// TwinCAT 3 PLC project Plc
// Title: CHALET_XPlanar
// Company: Beckhoff CH
// ProjectVersion: 5.8.1
// ProgramVersion: 3.1.4023.0
// libraries:
//   CHALET_BaseComponents, * (Beckhoff CH)
//   CHALET_Nc, * (Beckhoff CH)
//   Tc2_EtherCAT, * (Beckhoff Automation GmbH)
//   Tc2_Math, * (Beckhoff Automation GmbH)
//   Tc2_Standard, * (Beckhoff Automation GmbH)
//   Tc2_System, * (Beckhoff Automation GmbH)
//   Tc2_Utilities, * (Beckhoff Automation GmbH)
//   Tc3_EventLogger, * (Beckhoff Automation GmbH)
//   Tc3_Mc3Definitions, * (Beckhoff Automation GmbH)
//   Tc3_Mc3PlanarMotion, * (Beckhoff Automation GmbH)
//   Tc3_Module, * (Beckhoff Automation GmbH)
//   Tc3_Physics, * (Beckhoff Automation GmbH)
//   Tc3_XPlanarUtility, * (Beckhoff Automation GmbH)
// project tree:
//   COMPONENTs/Environment/ I_XP_Enviroment_PLC.TcIO, FB_XP_Environment.TcPOU, I_XP_Environment.TcIO
//   COMPONENTs/Feedback/ FB_XP_Feedback.TcPOU, I_XP_Feedback.TcIO, ST_PlanarObjectInfoEx.TcDUT
//   COMPONENTs/Mover/ FB_XP_Mover.TcPOU, I_XP_Mover.TcIO, I_XP_Mover_PLC.TcIO
//   COMPONENTs/Mover/ProductData/ FB_XP_ProductData.TcPOU, I_XP_ProductData.TcIO
//   COMPONENTs/Optional/Casting/ ToXpMover.TcPOU, ToXpStation.TcPOU (not stored), ToXpTrack.TcPOU
//   COMPONENTs/Optional/Trigger/ FB_XP_Trigger.TcPOU, I_XP_Trigger.TcIO
//   COMPONENTs/Optional/Zone/ FB_XP_SoretedListOfMover.TcPOU, I_XP_Zone.TcIO
//   COMPONENTs/Path/ FB_XP_Path.TcPOU, I_XP_Path.TcIO
//   COMPONENTs/Stationen/A-Star-Node/ FB_AStarNode.TcPOU, I_PathAStarNode.TcIO
//   COMPONENTs/Stationen/ FB_XP_Station.TcPOU, I_XP_Station.TcIO, I_XP_Station_PLC.TcIO
//   COMPONENTs/Group/ FB_XP_Group.TcPOU, I_XP_Group.TcIO
//   COMPONENTs/System/ FB_XP_System.TcPOU, I_XP_System_PLC.TcIO, I_XP_System_Registration.TcIO
//   COMPONENTs/Track/ FB_XP_Track.TcPOU, I_XP_Track.TcIO, I_XP_Track_PLC.TcIO
//   FUNCTIONs/ F_DistXYVectors.TcPOU, F_Vector_Multiplication.TcPOU, F_Vector_Subtraction.TcPOU, F_GetDistToPosModulo.TcPOU, F_InLimitTest.TcPOU, F_RotatePositionXY.TcPOU, F_Vector_Addition.TcPOU
//   / XPlanarParameterlist.TcGVL

// ---- COMPONENTs/Feedback/ST_PlanarObjectInfoEx.TcDUT
TYPE ST_PlanarObjectInfoEx EXTENDS Tc3_Mc3PlanarMotion.PlanarObjectInfo :
STRUCT
	ipObject : I_CH_Object;
END_STRUCT
END_TYPE

// ---- XPlanarParameterlist.TcGVL
{attribute 'qualified_only'}
VAR_GLOBAL CONSTANT 
	(*After the system init, this is the first station that is approached.
	 Can be used, for example, to send all movers to the “Unload” station first 
	 The default value is “not defined” so the movers remain in the closest station and wait for a valid destination*)
	S_MOVER_TARGED_INIT : STRING := 'not defined';	
	
	(*Only if enabled, mover take over "VelocytiAtExit" of passed station*)	
	B_STATIONS_OVERRIDE_MOVER_DYN_CONSTRAINT : BOOL := FALSE;
	
	(* Automatic generation of missing auxiliary stations on the track. 
	In order to clearly control the route of a mover, for example, when splitting a track into two tracks, an auxiliary station is created on both tracks. 
	The mover must pass this auxiliary station. It moves to it and crosses over as soon as the switch point is passed. 
	This auxiliary station cannot hold a mover (queue size 0) *)
	B_AUTOMATIC_GENARATE_HELPER_STATIONS : BOOL := TRUE;
	
	(*Minimum gap center to center on track [mm] *)
	F_MOVER_MINIMUM_GAP_ON_TRACK : LREAL := 100.0;
	
	(*Default gap center to center on track. Each station can override this gap[mm] *)
	F_GAP_DEFAULT: LREAL := 120.0;
	
	(*Determine the absolute C-rotation of the mover when starting up. Requires an “APM9001-0000-4xxx | XPlanar-ID-Bumper”. *)
	B_GET_MOVER_ORIENTATION : BOOL := FALSE;	
	B_ID_BUMPER_INSTALLED : BOOL := TRUE;
	
	(*Read mover ID when starting up. Requires an “APM9001-0000-4xxx | XPlanar-ID-Bumper”. *)
	B_GET_MOVER_ID : BOOL := FALSE;	
	
	//Quick stop on disable.
	//TRUE = The mover stops immediately AT the current position
	//FALSE = The mover cancels the superimposed ExternalSetpoint movement and returns to the track with maximum dynamic. -> Like a rubber band
	B_QUICKSTOP_ON_DISABLING : BOOL := TRUE;
	
	//When the system is enabled, the system checks which movers are actually present. 
	//Any movers that are not present are moved forward to the “NotPresent” list
	B_AUTOMATICALLY_REMOVE_NOT_PRESENT_MOVER_AT_ENABLING : BOOL := TRUE;	
	
	(*Add envirement to groupe during enabling *)
	B_ADD_ENVIROMENT_TO_GROUP : BOOL := TRUE;	
					
	(*Add tracks to groupe during enabling *)
	B_ADD_TRACKS_TO_GROUP : BOOL := FALSE;	
					
	(*Add movers to groupe during enabling *)
	B_ADD_MOVERS_TO_GROUP : BOOL := FALSE;	
					
	//Velocity during enabling move on track. 0=Default
	F_ENABLING_ON_TRACK_VELOCITY	: LREAL := 0;
	
	(*Acc-/Deceleration during enabling move on track. 0=Default*)
	F_ENABLING_ON_TRACK_ACC_DEC		: LREAL := 0;
	
	(*This value as a Station.Filter allows all movers of any target*)
	S_ANY_STATION_NAME : STRING := '';
	
	//TRUE = Use inside PLC the track name from the TcCom Track Object. If FALSE overwride TcCom Track object with instance name
	B_TRACK_NAME_TACKOVER_FROM_TRACK_OBJECT : BOOL := TRUE;
	
	//If a single-cell sequence step takes longer than this time when enabling the entire system, an error is generated and the enabling is aborted
	F_TIMEOUT_ERROR_ENABLING : LREAL := 30.0; //[s]
	
	(*The movers are only sent to the next free station on the way to the destination. 
	The distance in mm can be specified here to indicate how much further away the new move command can already be sent.  *)
	F_DIST_SET_NEW_MOVE_CMD_BEFORE_REACHING_PARENT_STATION : LREAL := 200.0;
	
	(*max tracks after a track switch *)
	N_MAX_STATIONS_AHEAD_OR_BEHIND : UINT := 20;	
	
	(*A mover must leave the station immediately when the ‘SendMoversToStation’ method is called. The station is then available again.
	Otherwise, if no destination station is available, the mover waits in the station.*)
	B_MOVER_MUST_LEAVE_STATION_AT_SET_NEW_TARGED : BOOL := TRUE;
	
	(*0: Indicates no or invalid information, e.g. no connection or component not yet ready. 
	1: The Planar Mover interprets the given dynamic limits in a one-dimensional fashion, with respect to the track's arclength. This way, the maximum velocity is aimed at even in curves. 
	2: The maximal velocity in curves is reduced to not exceed the maximum x,y radial acceleration there. Produces the same behavior as the None mode when on a straight track. 	*)
	N_SELECT_MODE_HOW_DYNAMIC_IS_PLANED_ON_TRACK : UINT := 2;
	
	(*Indicates the way in which gap control is done on track.
	1:The Planar Mover keeps a distance to its neighbours on track that is at least the sum of gap and stop distance.
	2:The Planar Mover keeps a distance to its neighbours on track that is at least the gap.*)
	N_GAP_MODE_ON_TRACK : UINT := 2;
	
	(* How many elements (point, line or arc) does the most complex track have? *)
	N_MAX_GEOMETRIC_ELEMENTS_PER_TRACK : UINT := 20;
END_VAR

// ---- COMPONENTs/Environment/I_XP_Enviroment_PLC.TcIO
INTERFACE I_XP_Enviroment_PLC EXTENDS I_CH_Object

{attribute 'monitoring':='call'}
(* If Enable, the movers are checked for collisions with each other.
Warning and error can have their own size offsets.
The error leads to a stop with higher dynamics.
In simulation, an error does not lead to a stop *)
PROPERTY CollisionCheck : BOOL
GET
END_GET
SET
END_SET
END_PROPERTY

{attribute 'monitoring':='call'}
//Offset on the mover dimension from the MC3 mover object [mm] ;
// >0 menas the warning is earlier
PROPERTY MoverCollisionOffsetError : LREAL
GET
END_GET
SET
END_SET
END_PROPERTY

{attribute 'monitoring':='call'}
//Offset on the mover dimension from the MC3 mover object [mm] ;
// >0 menas the warning is earlier
PROPERTY MoverCollisionOffsetWarning : LREAL
GET
END_GET
SET
END_SET
END_PROPERTY

{attribute 'monitoring':='call'}
//Enumeration MoverDetectionStatus
PROPERTY MoverDetectionStatus : MoverDetectionStatus
GET
END_GET
END_PROPERTY

{attribute 'monitoring':='call'}
//Object ID of the IoXPlanar processing unit
PROPERTY ProcessingUnitOID : OTCID
GET
END_GET
END_PROPERTY

{attribute 'monitoring':='call'}
//Interface to CHALET system to which this object belongs
PROPERTY System : I_XP_System_PLC
GET
END_GET
END_PROPERTY

END_INTERFACE

// ---- COMPONENTs/Feedback/I_XP_Feedback.TcIO
INTERFACE I_XP_Feedback EXTENDS CHALET_BaseComponents.I_CH_Feedback

{attribute 'monitoring':='call'}
(* Indicates which object one would collide with. *)
PROPERTY ObjectInfo : REFERENCE TO PlanarObjectInfo
GET
END_GET
SET
END_SET
END_PROPERTY

{attribute 'monitoring':='call'}
(* Indicates which object one would collide with. *)
PROPERTY ObjectInfoEx : REFERENCE TO ST_PlanarObjectInfoEx
GET
END_GET
SET
END_SET
END_PROPERTY

END_INTERFACE

// ---- COMPONENTs/Mover/I_XP_Mover.TcIO
INTERFACE I_XP_Mover  EXTENDS I_CH_Object

{attribute 'monitoring':='call'}
(* Provides the current planar mover setpoint XYZABC [mm/s²] *)
PROPERTY AccelerationSet : REFERENCE TO MoverVector
GET
END_GET
END_PROPERTY

METHOD AddToGroup : HRESULT
VAR_INPUT
	iGroup : I_XP_Group;
END_VAR
END_METHOD

{attribute 'monitoring':='call'}
(* C coordinate modulus set in MC3-Planar Mover[°] *)
PROPERTY CAxisModulo : LREAL
GET
END_GET
END_PROPERTY

{attribute 'monitoring':='call'}
PROPERTY CurrentTrack : I_XP_Track
GET
END_GET
END_PROPERTY

METHOD Disable : HRESULT
VAR_INPUT
END_VAR
END_METHOD

//This method is called when the system is disabled. Links are deleted as they may no longer be valid
METHOD Disassemble : HRESULT
VAR_INPUT
END_VAR
END_METHOD

{attribute 'monitoring':='call'}
PROPERTY DistToParentStation : LREAL //Distance to the responsible parent station [mm]
GET
END_GET
END_PROPERTY

METHOD DistToTrack : LREAL
VAR_INPUT
	iTrack : I_XP_Track;
END_VAR
END_METHOD

PROPERTY DynConstraint : REFERENCE TO DynamicConstraint_Container
GET
END_GET
END_PROPERTY

METHOD Enable : HRESULT
VAR_INPUT
END_VAR
END_METHOD

{attribute 'monitoring':='call'}
//operational and position control active(hovering)
PROPERTY Enabled : BOOL
GET
END_GET
END_PROPERTY

{attribute 'OPC.UA.DA.Property' := '1'}
{attribute 'monitoring':='call'}
PROPERTY Feedback : I_XP_Feedback
GET
END_GET
END_PROPERTY

METHOD Halt : HRESULT
VAR_INPUT
END_VAR
END_METHOD

METHOD JoinTrack : HRESULT
VAR_INPUT
	iTrack : I_XP_Track;
END_VAR
END_METHOD

{attribute 'monitoring':='call'}
PROPERTY LastCmdTargetGap : LREAL
GET
END_GET
END_PROPERTY

{attribute 'monitoring':='call'}
PROPERTY LastCmdTargetPosition : LREAL
GET
END_GET
END_PROPERTY

{attribute 'monitoring':='call'}
PROPERTY LastCmdTargetTrack: I_XP_Track
GET
END_GET
END_PROPERTY

{attribute 'monitoring':='call'}
//This was the last valid (system enabled) parent station of the mover
PROPERTY LastValidParentStation : I_XP_Station;
GET
END_GET
END_PROPERTY

{attribute 'monitoring':='call'}
//This was the last valid (system enabled) actual  position of the mover
PROPERTY LastValidPositionOnTrack : LREAL
GET
END_GET
END_PROPERTY

{attribute 'monitoring':='call'}
//This was the last valid (system enabled) actual  position of the mover
PROPERTY LastValidPositionXYZABC : REFERENCE TO MoverVector
GET
END_GET
END_PROPERTY

{attribute 'monitoring':='call'}
//This was the last valid (system enabled) actual  position of the mover
PROPERTY LastValidTrack : I_XP_Track;
GET
END_GET
END_PROPERTY

//The mover returns to its SetPos. The force of the Z, A and B axis is slowly increased.
METHOD LiftFromUnknownLevel : HRESULT
VAR_INPUT
END_VAR
END_METHOD

(* The mover is lowered. The target height is unknown. The force from the Z, A and B axles is then reduced to a minimum. X, Y and C still remain active.
   This function can be used, for example, to place the mover in a holder.  *)
METHOD LowerToUnknownLevel : HRESULT
VAR_INPUT
END_VAR
END_METHOD

{attribute 'monitoring':='call'}
PROPERTY Mapped : BOOL //Project is mapped to MC (McToPlc and PlcToMc)
GET
END_GET
END_PROPERTY

{attribute 'monitoring':='call'}
PROPERTY Mode : MC_PLANAR_MOVER_COMMAND_MODE
GET
END_GET
END_PROPERTY

METHOD MoveA : HRESULT
VAR_INPUT
	fPosition : LREAL;
END_VAR
END_METHOD

METHOD MoveB : HRESULT
VAR_INPUT
	fPosition : LREAL;
END_VAR
END_METHOD

METHOD MoveC : HRESULT
VAR_INPUT
	fPosition : LREAL;
	
	(* Addition turns to move in modulo movement (positive or negative). *)
	additionalTurns : UDINT := 0;
	
	(* Direction in which the target is approached. *)
	direction : Tc3_Mc3Definitions.MC_DIRECTION := Tc3_Mc3Definitions.MC_DIRECTION.mcDirectionNonModulo;
END_VAR
END_METHOD

METHOD MoveOnTrack : HRESULT
VAR_INPUT
	ipTrack : I_XP_Track;
	fPosition : LREAL;
	fGap : LREAL;
END_VAR
END_METHOD

METHOD MoveOnTrack_ShortestWay : HRESULT
VAR_INPUT
	ipTrack : I_XP_Track;
	fPosition : LREAL;
	fGap : LREAL;
END_VAR
END_METHOD

METHOD MoveOnTrackToStation : HRESULT
VAR_INPUT
	ipStation : I_XP_Station;
	fGap : LREAL;
END_VAR
END_METHOD

{attribute 'monitoring':='call'}
(* Height that is used for internal collision checks.[mm] *)
PROPERTY MoverHeight : LREAL
GET
END_GET
END_PROPERTY

{attribute 'monitoring':='call'}
//Mover could not be detected or was removed from the system
PROPERTY MoverIsNotPresent : BOOL
GET
END_GET
END_PROPERTY

{attribute 'monitoring':='call'}
(* Width that is used for internal collision checks.[mm] *)
PROPERTY MoverWidth : LREAL
GET
END_GET
END_PROPERTY

METHOD MoveXY : HRESULT
VAR_INPUT
	fPosition_X : LREAL;
	fPosition_Y : LREAL;
END_VAR
END_METHOD

METHOD MoveZ : HRESULT
VAR_INPUT
	fPosition : LREAL;
END_VAR
END_METHOD

{attribute 'monitoring':='call'}
//Unique object ID
PROPERTY OID : OTCID
GET
END_GET
END_PROPERTY

{attribute 'monitoring':='call'}
PROPERTY ParentStation : I_XP_Station
GET
END_GET
SET
END_SET
END_PROPERTY

{attribute 'monitoring':='call'}
PROPERTY PlanarMover : REFERENCE TO MC_PlanarMover
GET
END_GET
END_PROPERTY

{attribute 'monitoring':='call'}
(* Contains the information of the Planar Mover passed from MC to PLC. XYZABC [mm] *)
PROPERTY PositionAct : REFERENCE TO MoverVector
GET
END_GET
END_PROPERTY

{attribute 'monitoring':='call'}
PROPERTY PositionOnTrack : LREAL
GET
END_GET
END_PROPERTY

{attribute 'monitoring':='call'}
(* Provides the current planar mover setpoint XYZABC [mm] *)
PROPERTY PositionSet : REFERENCE TO MoverVector
GET
END_GET
END_PROPERTY

METHOD RemoveFromGroup : HRESULT
END_METHOD

METHOD Reset : HRESULT
VAR_INPUT
END_VAR
END_METHOD

{attribute 'monitoring':='call'}
//Complete route from last parent to active parent station
PROPERTY RouteComplete : I_CH_List
GET
END_GET
END_PROPERTY

{attribute 'monitoring':='call'}
//Remaining route to the parent
PROPERTY RouteRemaining: I_CH_List
GET
END_GET
END_PROPERTY

//done segments can be transferred here. these are removed from the remaining route
METHOD RouteSegmentDone : BOOL
VAR_INPUT
	ipPathDone : I_XP_Path;
END_VAR
END_METHOD

METHOD SetDynConstraint_A : BOOL //Dynamic constraints for individual coordinates.
VAR_INPUT
    V : MC_LREAL; //equivalent to data type LREAL + MC_DEFAULT, MC_MAXIMUM
    A : MC_LREAL; //equivalent to data type LREAL + MC_DEFAULT, MC_MAXIMUM
    D : MC_LREAL; //equivalent to data type LREAL + MC_DEFAULT, MC_MAXIMUM
    J : MC_LREAL; //equivalent to data type LREAL + MC_DEFAULT, MC_MAXIMUM
END_VAR
END_METHOD

METHOD SetDynConstraint_B : BOOL //Dynamic constraints for individual coordinates.
VAR_INPUT
    V : MC_LREAL; //equivalent to data type LREAL + MC_DEFAULT, MC_MAXIMUM
    A : MC_LREAL; //equivalent to data type LREAL + MC_DEFAULT, MC_MAXIMUM
    D : MC_LREAL; //equivalent to data type LREAL + MC_DEFAULT, MC_MAXIMUM
    J : MC_LREAL; //equivalent to data type LREAL + MC_DEFAULT, MC_MAXIMUM
END_VAR
END_METHOD

METHOD SetDynConstraint_C : BOOL //Dynamic constraints for individual coordinates.
VAR_INPUT
    V : MC_LREAL; //equivalent to data type LREAL + MC_DEFAULT, MC_MAXIMUM
    A : MC_LREAL; //equivalent to data type LREAL + MC_DEFAULT, MC_MAXIMUM
    D : MC_LREAL; //equivalent to data type LREAL + MC_DEFAULT, MC_MAXIMUM
    J : MC_LREAL; //equivalent to data type LREAL + MC_DEFAULT, MC_MAXIMUM
END_VAR
END_METHOD

METHOD SetDynConstraint_Path : BOOL //One dimensional dynamic constraint along the XY-components of a path, ignoring non-tangential effects.
VAR_INPUT
    V : MC_LREAL; //equivalent to data type LREAL + MC_DEFAULT, MC_MAXIMUM
    A : MC_LREAL; //equivalent to data type LREAL + MC_DEFAULT, MC_MAXIMUM
    D : MC_LREAL; //equivalent to data type LREAL + MC_DEFAULT, MC_MAXIMUM
    J : MC_LREAL; //equivalent to data type LREAL + MC_DEFAULT, MC_MAXIMUM
END_VAR
END_METHOD

METHOD SetDynConstraint_X : BOOL //Dynamic constraints for individual coordinates.
VAR_INPUT
    V : MC_LREAL; //equivalent to data type LREAL + MC_DEFAULT, MC_MAXIMUM
    A : MC_LREAL; //equivalent to data type LREAL + MC_DEFAULT, MC_MAXIMUM
    D : MC_LREAL; //equivalent to data type LREAL + MC_DEFAULT, MC_MAXIMUM
    J : MC_LREAL; //equivalent to data type LREAL + MC_DEFAULT, MC_MAXIMUM
END_VAR
END_METHOD

METHOD SetDynConstraint_Y : BOOL //Dynamic constraints for individual coordinates.
VAR_INPUT
    V : MC_LREAL; //equivalent to data type LREAL + MC_DEFAULT, MC_MAXIMUM
    A : MC_LREAL; //equivalent to data type LREAL + MC_DEFAULT, MC_MAXIMUM
    D : MC_LREAL; //equivalent to data type LREAL + MC_DEFAULT, MC_MAXIMUM
    J : MC_LREAL; //equivalent to data type LREAL + MC_DEFAULT, MC_MAXIMUM
END_VAR
END_METHOD

METHOD SetDynConstraint_Z : BOOL //Dynamic constraints for individual coordinates.
VAR_INPUT
    V : MC_LREAL; //equivalent to data type LREAL + MC_DEFAULT, MC_MAXIMUM
    A : MC_LREAL; //equivalent to data type LREAL + MC_DEFAULT, MC_MAXIMUM
    D : MC_LREAL; //equivalent to data type LREAL + MC_DEFAULT, MC_MAXIMUM
    J : MC_LREAL; //equivalent to data type LREAL + MC_DEFAULT, MC_MAXIMUM
END_VAR
END_METHOD

METHOD SetRouteToParent : HRESULT
VAR_INPUT
	ipRoute : I_CH_LIST;
END_VAR
END_METHOD

{attribute 'monitoring':='call'}
(* Velocity is zero *)
PROPERTY Standstill : BOOL
GET
END_GET
END_PROPERTY

METHOD StopExternalSetpoint : HRESULT
VAR_INPUT
END_VAR
END_METHOD

{attribute 'monitoring':='call'}
PROPERTY TargetStation : String
GET
END_GET
SET
END_SET
END_PROPERTY

{attribute 'monitoring':='call'}
PROPERTY UtilityMcMover : Tc3_XPlanarUtility.I_McPlanarMover
GET
END_GET
END_PROPERTY

PROPERTY UtilityTcIoMover : Tc3_XPlanarUtility.I_TcIoXPlanarMover
GET
END_GET
END_PROPERTY

{attribute 'monitoring':='call'}
(* Provides the current planar mover act XYZABC [mm/s] *)
PROPERTY VelocityAct : REFERENCE TO MoverVector
GET
END_GET
END_PROPERTY

{attribute 'monitoring':='call'}
(* Provides the current planar mover setpoint XYZABC [mm/s] *)
PROPERTY VelocitySet : REFERENCE TO MoverVector
GET
END_GET
END_PROPERTY

END_INTERFACE

// ---- COMPONENTs/Mover/I_XP_Mover_PLC.TcIO
INTERFACE I_XP_Mover_PLC EXTENDS I_CH_Object

{attribute 'monitoring':='call'}
(* Provides the current planar mover setpoint XYZABC [mm/s²] *)
PROPERTY AccelerationSet : REFERENCE TO MoverVector
GET
END_GET
END_PROPERTY

{attribute 'monitoring':='call'}
PROPERTY  AxisExtSetpointA : CHALET_Nc.I_NcAxis_PLC
GET
END_GET
END_PROPERTY

{attribute 'monitoring':='call'}
PROPERTY AxisExtSetpointB : CHALET_Nc.I_NcAxis_PLC
GET
END_GET
END_PROPERTY

{attribute 'monitoring':='call'}
PROPERTY AxisExtSetpointC : CHALET_Nc.I_NcAxis_PLC
GET
END_GET
END_PROPERTY

{attribute 'monitoring':='call'}
PROPERTY  AxisExtSetpointX : CHALET_Nc.I_NcAxis_PLC
GET
END_GET
END_PROPERTY

{attribute 'monitoring':='call'}
PROPERTY AxisExtSetpointY : CHALET_Nc.I_NcAxis_PLC
GET
END_GET
END_PROPERTY

{attribute 'monitoring':='call'}
PROPERTY AxisExtSetpointZ : CHALET_Nc.I_NcAxis_PLC
GET
END_GET
END_PROPERTY

{attribute 'monitoring':='call'}
(* C coordinate modulus set in MC3-Planar Mover[°] *)
PROPERTY CAxisModulo : LREAL
GET
END_GET
END_PROPERTY

{attribute 'monitoring':='call'}
(* Indicates the command mode of an enabled PlanarMover, i.e. how setpoints are currently produced. *)
PROPERTY CommandMode : MC_PLANAR_MOVER_COMMAND_MODE
GET
END_GET
END_PROPERTY

{attribute 'monitoring':='call'}
PROPERTY CurrentTrack : I_XP_Track
GET
END_GET
END_PROPERTY

{attribute 'monitoring':='call'}
PROPERTY DistToParentStation : LREAL //Distance to the responsible parent station [mm]
GET
END_GET
END_PROPERTY

METHOD DistToTrack : LREAL
VAR_INPUT
	iTrack : I_XP_Track;
END_VAR
END_METHOD

PROPERTY DynConstraint : REFERENCE TO DynamicConstraint_Container
GET
END_GET
END_PROPERTY

{attribute 'monitoring':='call'}
//operational and position control active(hovering)
PROPERTY Enabled : BOOL
GET
END_GET
END_PROPERTY

{attribute 'OPC.UA.DA.Property' := '1'}
{attribute 'monitoring':='call'}
PROPERTY Feedback : I_XP_Feedback
GET
END_GET
END_PROPERTY

METHOD Halt : HRESULT
VAR_INPUT
END_VAR
END_METHOD

METHOD JoinTrack : HRESULT
VAR_INPUT
	iTrack : I_XP_Track;
END_VAR
END_METHOD

{attribute 'monitoring':='call'}
(* Retruns lentgh of hypotenuse of the x and y error. (>=0[mm]) *)
PROPERTY LagDistanceXY : LREAL
GET
END_GET
END_PROPERTY

{attribute 'monitoring':='call'}
PROPERTY LastCmdTargetGap : LREAL
GET
END_GET
END_PROPERTY

{attribute 'monitoring':='call'}
PROPERTY LastCmdTargetPosition : LREAL
GET
END_GET
END_PROPERTY

{attribute 'monitoring':='call'}
PROPERTY LastCmdTargetTrack: I_XP_Track
GET
END_GET
END_PROPERTY

{attribute 'monitoring':='call'}
//This was the last valid (system enabled) parent station of the mover
PROPERTY LastValidParentStation : I_XP_Station;
GET
END_GET
END_PROPERTY

{attribute 'monitoring':='call'}
//This was the last valid (system enabled) actual  position of the mover
PROPERTY LastValidPositionOnTrack : LREAL
GET
END_GET
END_PROPERTY

{attribute 'monitoring':='call'}
//This was the last valid (system enabled) actual  position of the mover
PROPERTY LastValidPositionXYZABC : REFERENCE TO MoverVector
GET
END_GET
END_PROPERTY

{attribute 'monitoring':='call'}
//This was the last valid (system enabled) actual  position of the mover
PROPERTY LastValidTrack : I_XP_Track;
GET
END_GET
END_PROPERTY

//The mover returns to its SetPos. The force of the Z, A and B axis is slowly increased.
METHOD LiftFromUnknownLevel : HRESULT
VAR_INPUT
END_VAR
END_METHOD

(* The mover is lowered. The target height is unknown. The force from the Z, A and B axles is then reduced to a minimum. X, Y and C still remain active.
   This function can be used, for example, to place the mover in a holder.  *)
METHOD LowerToUnknownLevel : HRESULT
VAR_INPUT
END_VAR
END_METHOD

{attribute 'monitoring':='call'}
PROPERTY LUID : STRING //Locally unique identifier
GET
END_GET
END_PROPERTY

{attribute 'monitoring':='call'}
PROPERTY Mapped : BOOL //Project is mapped to MC (McToPlc and PlcToMc)
GET
END_GET
END_PROPERTY

METHOD MoveA : HRESULT
VAR_INPUT
	fPosition : LREAL;
END_VAR
END_METHOD

METHOD MoveB : HRESULT
VAR_INPUT
	fPosition : LREAL;
END_VAR
END_METHOD

METHOD MoveC : HRESULT
VAR_INPUT
	fPosition : LREAL;
	
	(* Addition turns to move in modulo movement (positive or negative). *)
	additionalTurns : UDINT := 0;
	
	(* Direction in which the target is approached. *)
	direction : Tc3_Mc3Definitions.MC_DIRECTION := Tc3_Mc3Definitions.MC_DIRECTION.mcDirectionNonModulo;
END_VAR
END_METHOD

METHOD MoveOnTrack : HRESULT
VAR_INPUT
	ipTrack : I_XP_Track;
	fPosition : LREAL;
	fGap : LREAL;
END_VAR
END_METHOD

METHOD MoveOnTrack_ShortestWay : HRESULT
VAR_INPUT
	ipTrack : I_XP_Track;
	fPosition : LREAL;
	fGap : LREAL;
END_VAR
END_METHOD

{attribute 'monitoring':='call'}
(* Height that is used for internal collision checks.[mm] *)
PROPERTY MoverHeight : LREAL
GET
END_GET
END_PROPERTY

{attribute 'monitoring':='call'}
//Mover could not be detected or was removed from the system
PROPERTY MoverIsNotPresent : BOOL
GET
END_GET
END_PROPERTY

{attribute 'monitoring':='call'}
(* Width that is used for internal collision checks.[mm] *)
PROPERTY MoverWidth : LREAL
GET
END_GET
END_PROPERTY

METHOD MoveXY : HRESULT
VAR_INPUT
	fPosition_X : LREAL;
	fPosition_Y : LREAL;
END_VAR
END_METHOD

METHOD MoveZ : HRESULT
VAR_INPUT
	fPosition : LREAL;
END_VAR
END_METHOD

{attribute 'monitoring':='call'}
//Unique object ID
PROPERTY OID : OTCID
GET
END_GET
END_PROPERTY

{attribute 'monitoring':='call'}
PROPERTY ParentStation : I_XP_Station
GET
END_GET
END_PROPERTY

{attribute 'monitoring':='call'}
PROPERTY PlanarMover : REFERENCE TO MC_PlanarMover
GET
END_GET
END_PROPERTY

{attribute 'monitoring':='call'}
(* Contains the information of the Planar Mover passed from MC to PLC. XYZABC [mm] *)
PROPERTY PositionAct : REFERENCE TO MoverVector
GET
END_GET
END_PROPERTY

{attribute 'monitoring':='call'}
PROPERTY PositionOnTrack : LREAL
GET
END_GET
END_PROPERTY

{attribute 'monitoring':='call'}
(* Provides the current planar mover setpoint XYZABC [mm] *)
PROPERTY PositionSet : REFERENCE TO MoverVector
GET
END_GET
END_PROPERTY

{attribute 'monitoring':='call'}
PROPERTY PUBLIC ProductData : I_XP_ProductData
GET
END_GET
SET
END_SET
END_PROPERTY

{attribute 'monitoring':='call'}
//Complete route from last parent to active parent station
PROPERTY RouteComplete : I_CH_List
GET
END_GET
END_PROPERTY

{attribute 'monitoring':='call'}
//Remaining route to the parent
PROPERTY RouteRemaining: I_CH_List
GET
END_GET
END_PROPERTY

//done segments can be transferred here. these are removed from the remaining route
METHOD RouteSegmentDone : BOOL
VAR_INPUT
	ipPathDone : I_XP_Path;
END_VAR
END_METHOD

METHOD SetDynConstraint_A : BOOL //Dynamic constraints for individual coordinates.
VAR_INPUT
    V : MC_LREAL; //equivalent to data type LREAL + MC_DEFAULT, MC_MAXIMUM
    A : MC_LREAL; //equivalent to data type LREAL + MC_DEFAULT, MC_MAXIMUM
    D : MC_LREAL; //equivalent to data type LREAL + MC_DEFAULT, MC_MAXIMUM
    J : MC_LREAL; //equivalent to data type LREAL + MC_DEFAULT, MC_MAXIMUM
END_VAR
END_METHOD

METHOD SetDynConstraint_B : BOOL //Dynamic constraints for individual coordinates.
VAR_INPUT
    V : MC_LREAL; //equivalent to data type LREAL + MC_DEFAULT, MC_MAXIMUM
    A : MC_LREAL; //equivalent to data type LREAL + MC_DEFAULT, MC_MAXIMUM
    D : MC_LREAL; //equivalent to data type LREAL + MC_DEFAULT, MC_MAXIMUM
    J : MC_LREAL; //equivalent to data type LREAL + MC_DEFAULT, MC_MAXIMUM
END_VAR
END_METHOD

METHOD SetDynConstraint_C : BOOL //Dynamic constraints for individual coordinates.
VAR_INPUT
    V : MC_LREAL; //equivalent to data type LREAL + MC_DEFAULT, MC_MAXIMUM
    A : MC_LREAL; //equivalent to data type LREAL + MC_DEFAULT, MC_MAXIMUM
    D : MC_LREAL; //equivalent to data type LREAL + MC_DEFAULT, MC_MAXIMUM
    J : MC_LREAL; //equivalent to data type LREAL + MC_DEFAULT, MC_MAXIMUM
END_VAR
END_METHOD

METHOD SetDynConstraint_Path : BOOL //One dimensional dynamic constraint along the XY-components of a path, ignoring non-tangential effects.
VAR_INPUT
    V : MC_LREAL; //equivalent to data type LREAL + MC_DEFAULT, MC_MAXIMUM
    A : MC_LREAL; //equivalent to data type LREAL + MC_DEFAULT, MC_MAXIMUM
    D : MC_LREAL; //equivalent to data type LREAL + MC_DEFAULT, MC_MAXIMUM
    J : MC_LREAL; //equivalent to data type LREAL + MC_DEFAULT, MC_MAXIMUM
END_VAR
END_METHOD

METHOD SetDynConstraint_X : BOOL //Dynamic constraints for individual coordinates.
VAR_INPUT
    V : MC_LREAL; //equivalent to data type LREAL + MC_DEFAULT, MC_MAXIMUM
    A : MC_LREAL; //equivalent to data type LREAL + MC_DEFAULT, MC_MAXIMUM
    D : MC_LREAL; //equivalent to data type LREAL + MC_DEFAULT, MC_MAXIMUM
    J : MC_LREAL; //equivalent to data type LREAL + MC_DEFAULT, MC_MAXIMUM
END_VAR
END_METHOD

METHOD SetDynConstraint_Y : BOOL //Dynamic constraints for individual coordinates.
VAR_INPUT
    V : MC_LREAL; //equivalent to data type LREAL + MC_DEFAULT, MC_MAXIMUM
    A : MC_LREAL; //equivalent to data type LREAL + MC_DEFAULT, MC_MAXIMUM
    D : MC_LREAL; //equivalent to data type LREAL + MC_DEFAULT, MC_MAXIMUM
    J : MC_LREAL; //equivalent to data type LREAL + MC_DEFAULT, MC_MAXIMUM
END_VAR
END_METHOD

METHOD SetDynConstraint_Z : BOOL //Dynamic constraints for individual coordinates.
VAR_INPUT
    V : MC_LREAL; //equivalent to data type LREAL + MC_DEFAULT, MC_MAXIMUM
    A : MC_LREAL; //equivalent to data type LREAL + MC_DEFAULT, MC_MAXIMUM
    D : MC_LREAL; //equivalent to data type LREAL + MC_DEFAULT, MC_MAXIMUM
    J : MC_LREAL; //equivalent to data type LREAL + MC_DEFAULT, MC_MAXIMUM
END_VAR
END_METHOD

METHOD SetRouteToParent : HRESULT
VAR_INPUT
	ipRoute : I_CH_LIST;
END_VAR
END_METHOD

{attribute 'monitoring':='call'}
(* Velocity is zero *)
PROPERTY Standstill : BOOL
GET
END_GET
END_PROPERTY

METHOD StartExternalSetpoint : HRESULT
END_METHOD

METHOD StopExternalSetpoint : HRESULT
VAR_INPUT
END_VAR
END_METHOD

{attribute 'monitoring':='call'}
//Interface to CHALET system to which this object belongs
PROPERTY System : I_XP_System_PLC
GET
END_GET
END_PROPERTY

{attribute 'monitoring':='call'}
PROPERTY TargetStation : STRING
GET
END_GET
SET
END_SET
END_PROPERTY

{attribute 'monitoring':='call'}
PROPERTY UtilityMcMover : Tc3_XPlanarUtility.I_McPlanarMover
GET
END_GET
END_PROPERTY

{attribute 'monitoring':='call'}
PROPERTY UtilityTcIoMover : Tc3_XPlanarUtility.I_TcIoXPlanarMover
GET
END_GET
END_PROPERTY

{attribute 'monitoring':='call'}
(* Provides the current planar mover act XYZABC [mm/s] *)
PROPERTY VelocityAct : REFERENCE TO MoverVector
GET
END_GET
END_PROPERTY

{attribute 'monitoring':='call'}
(* Provides the current planar mover setpoint XYZABC [mm/s] *)
PROPERTY VelocitySet : REFERENCE TO MoverVector
GET
END_GET
END_PROPERTY

END_INTERFACE

// ---- COMPONENTs/Mover/ProductData/I_XP_ProductData.TcIO
INTERFACE I_XP_ProductData EXTENDS __SYSTEM.IQueryInterface

{attribute 'monitoring':='call'}
PROPERTY LinkedMover : I_XP_Mover_PLC
GET
END_GET
END_PROPERTY

METHOD LinkToMover : BOOL //it is not necessary to call this method. This is already done internally
VAR_INPUT
	ipMoverPlc : I_XP_Mover_PLC;
END_VAR
END_METHOD

END_INTERFACE

// ---- COMPONENTs/Optional/Trigger/I_XP_Trigger.TcIO
INTERFACE I_XP_Trigger  EXTENDS __SYSTEM.IQueryInterface

{attribute 'monitoring':='call'}
PROPERTY AccocietedTrack : I_XP_Track
GET
END_GET
SET
END_SET
END_PROPERTY

{attribute 'monitoring':='call'}
PROPERTY HR : HRESULT
GET
END_GET
END_PROPERTY

PROPERTY ListOfMoversToCheck : I_CH_List
SET
END_SET
END_PROPERTY

{attribute 'monitoring':='call'}
PROPERTY MoverAtTrigger : I_XP_Mover
GET
END_GET
END_PROPERTY

{attribute 'monitoring':='call'}
PROPERTY MoverDetected : BOOL
GET
END_GET
END_PROPERTY

{attribute 'monitoring':='call'}
PROPERTY PositionOnTrack : LREAL
GET
END_GET
SET
END_SET
END_PROPERTY

{attribute 'monitoring':='call'}
PROPERTY TimeStamp : T_DCTIME64;
GET
END_GET
END_PROPERTY

{attribute 'monitoring':='call'}
PROPERTY TriggerDirection : Tc3_Mc3Definitions.MC_Direction
GET
END_GET
SET
END_SET
END_PROPERTY

END_INTERFACE

// ---- COMPONENTs/Optional/Zone/I_XP_Zone.TcIO
INTERFACE I_XP_Zone

{attribute 'monitoring':='call'}
PROPERTY CtsMoversInZone : UINT
GET
END_GET
END_PROPERTY

{attribute 'monitoring':='call'}
PROPERTY MoversInZone : REFERENCE TO ARRAY [0..(CHALET_BaseComponents.BaseParameterlist.MAX_OBJECTS-1)] OF I_XP_Mover_PLC // Return a sorted list of movers in this zone. Index 0 is the mover in Front.
GET
END_GET
END_PROPERTY

END_INTERFACE

// ---- COMPONENTs/Path/I_XP_Path.TcIO
INTERFACE I_XP_Path  EXTENDS I_CH_Object

METHOD DistanceToDestiantion : LREAL
VAR_INPUT
	ipTrack : I_XP_Track;
	fPosOnTrack : LREAL;
END_VAR
END_METHOD

{attribute 'monitoring':='call'}
PROPERTY Length : LREAL
GET
END_GET
SET
END_SET
END_PROPERTY

{attribute 'monitoring':='call'}
PROPERTY StationDestination : I_XP_Station
GET
END_GET
SET
END_SET
END_PROPERTY

{attribute 'monitoring':='call'}
PROPERTY StationStart  : I_XP_Station
GET
END_GET
SET
END_SET
END_PROPERTY

{attribute 'monitoring':='call'}
PROPERTY TracksUsed : REFERENCE TO FB_CH_List
GET
END_GET
END_PROPERTY

END_INTERFACE

// ---- COMPONENTs/Stationen/A-Star-Node/I_PathAStarNode.TcIO
INTERFACE I_PathAStarNode EXTENDS I_CH_Object

{attribute 'monitoring':='call'}
PROPERTY PathLength : LREAL
GET
END_GET
END_PROPERTY

{attribute 'monitoring':='call'}
PROPERTY RouteUsedToNode : REFERENCE TO FB_CH_List
GET
END_GET
END_PROPERTY

{attribute 'monitoring':='call'}
PROPERTY Station : I_XP_Station
GET
END_GET
SET
END_SET
END_PROPERTY

END_INTERFACE

// ---- COMPONENTs/Stationen/I_XP_Station.TcIO
INTERFACE I_XP_Station EXTENDS I_CH_Object

{attribute 'monitoring':='call'}
//Track on which the station is located
PROPERTY AccocietedTrack : I_XP_Track
GET
END_GET
END_PROPERTY

METHOD AddMoverToQueue : HRESULT
VAR_INPUT
	ipMover : I_XP_Mover;
END_VAR
END_METHOD

{attribute 'monitoring':='call'}
//List of movers managed by this station
PROPERTY AssignedMovers : I_CH_List
GET
END_GET
END_PROPERTY

//Call this Methode whith seq 0->100, and wait each step until S_OK is returned
METHOD Configure : HRESULT
VAR_INPUT
	nSeq : UINT; //0->100
END_VAR
END_METHOD

{attribute 'monitoring':='call'}
PROPERTY CtsEmptySpaceInQueue : UDINT
GET
END_GET
END_PROPERTY

{attribute 'monitoring':='call'}
PROPERTY CtsMoversInQueue : UDINT
GET
END_GET
END_PROPERTY

{attribute 'monitoring':='call'}
(*[mm]
As soon as the mover is closer than this distance, the mover can be sent on to the next one if necessary.
This is the distance from the station to the end of the track or the shortest path to this station. Depending on which is closer. This is to ensure that the mover can no longer be overhauled.
This proberty can make the internal calculated distance smaller but not larger
Recalculated each disable/enable of the system*)
PROPERTY DecisionDistance : LREAL
GET
END_GET
SET
END_SET
END_PROPERTY

METHOD DeleteMoversQueue : HRESULT
VAR_INPUT
END_VAR
END_METHOD

//This method is called when the system is disabled. Links are deleted as they may no longer be valid
METHOD Disassemble : HRESULT
VAR_INPUT
END_VAR
END_METHOD

{attribute 'monitoring':='call'}
PROPERTY Filter : STRING
GET
END_GET
SET
END_SET
END_PROPERTY

{attribute 'monitoring':='call'}
PROPERTY MoverAccAtExit : MC_LREAL //[mm/s² on Track] Every mover that leaves or passes the station gets this new acceleration as a target.
GET
END_GET
END_PROPERTY

{attribute 'monitoring':='call'}
PROPERTY MoverDecAtExit : MC_LREAL //[mm/s² on Track] Every mover that leaves or passes the station gets this new deceleration as a target.
GET
END_GET
END_PROPERTY

{attribute 'monitoring':='call'}
//[mm] Every mover that leaves or passes the station gets this new gap as a target.
PROPERTY MoverGapAtExit : LREAL
GET
END_GET
SET
END_SET
END_PROPERTY

{attribute 'monitoring':='call'}
PROPERTY MoverQueueSize : UINT
GET
END_GET
END_PROPERTY

{attribute 'monitoring':='call'}
PROPERTY MoversInPlace : BOOL
GET
END_GET
END_PROPERTY

{attribute 'monitoring':='call'}
PROPERTY MoverVelocityAtExit : MC_LREAL //[mm/s on Track] Every mover that leaves or passes the station gets this new velocity as a target.
GET
END_GET
END_PROPERTY

{attribute 'monitoring':='call'}
//List of paths that lead to stations before this station
PROPERTY PathsAhead : I_CH_List
GET
END_GET
END_PROPERTY

{attribute 'monitoring':='call'}
//List of paths that lead to stations behind this station
PROPERTY PathsBehinde : I_CH_List
GET
END_GET
END_PROPERTY

{attribute 'monitoring':='call'}
//[mm] from the beginning of the assigned track
PROPERTY PositionOnTrack : LREAL
GET
END_GET
END_PROPERTY

{attribute 'monitoring':='call'}
//Position on the assigned track
PROPERTY PositionOnTrackXY : REFERENCE TO PositionXY
GET
END_GET
END_PROPERTY

{attribute 'monitoring':='call'}
//Position on the assigned track
PROPERTY PositionOnTrackXYZABC : REFERENCE TO MoverVector
GET
END_GET
END_PROPERTY

{attribute 'monitoring':='call'}
//Planned position, not necessarily on the track
PROPERTY PositionXY : REFERENCE TO  PositionXY
GET
END_GET
END_PROPERTY

//The movers currently in this station must leave the station. 
//The movers actively search for a destination, but only leave if a new destination is available.
METHOD PushMoversOutOfStation : HRESULT
VAR_INPUT
END_VAR
END_METHOD

{attribute 'monitoring':='call'}
//prevent further movers from entering the station, 
//e.g. to prevent a collision. All movers that are already moving to reach this station will be stopped with a stop 
//and restarted with Ready True.
PROPERTY ReadyToRecvMovers : BOOL
GET
END_GET
END_PROPERTY

METHOD SendMoversToStation : I_CH_Feedback //All movers in the station are sent to this destination
VAR_INPUT
	sTargetStation: STRING;//unique station name or group of stations
END_VAR
END_METHOD

{attribute 'monitoring':='call'}
//List of stations before this station
PROPERTY StationsAhead : I_CH_List
GET
END_GET
END_PROPERTY

{attribute 'monitoring':='call'}
//List of stations behinde this station
PROPERTY StationsBehinde : I_CH_List
GET
END_GET
END_PROPERTY

{attribute 'monitoring':='call'}
PROPERTY TargetGroupe : STRING
GET
END_GET
END_PROPERTY

METHOD Update : HRESULT
VAR_INPUT
END_VAR
END_METHOD

END_INTERFACE

// ---- COMPONENTs/Stationen/I_XP_Station_PLC.TcIO
INTERFACE I_XP_Station_PLC EXTENDS I_CH_Object

{attribute 'monitoring':='call'}
//Track on which the station is located
PROPERTY AccocietedTrack : I_XP_Track
GET
END_GET
END_PROPERTY

{attribute 'monitoring':='call'}
PROPERTY CtsEmptySpaceInQueue : UDINT
GET
END_GET
END_PROPERTY

{attribute 'monitoring':='call'}
PROPERTY CtsMoversInQueue : UDINT
GET
END_GET
END_PROPERTY

{attribute 'monitoring':='call'}
(*[mm]
As soon as the mover is closer than this distance, the mover can be sent on to the next one if necessary.
This is the distance from the station to the end of the track or the shortest path to this station. Depending on which is closer. This is to ensure that the mover can no longer be overhauled.
This proberty can make the internal calculated distance smaller but not larger
Recalculated each disable/enable of the system*)
PROPERTY DecisionDistance : LREAL
GET
END_GET
SET
END_SET
END_PROPERTY

{attribute 'monitoring':='call'}
PROPERTY Feedback : I_CH_Feedback
GET
END_GET
END_PROPERTY

{attribute 'monitoring':='call'}
//Filter content, movers with one of these targets may not approach or drive over the station
PROPERTY Filter : STRING
GET
END_GET
SET
END_SET
END_PROPERTY

{attribute 'monitoring':='call'}
PROPERTY LUID : STRING //Locally unique identifier
GET
END_GET
END_PROPERTY

{attribute 'monitoring':='call'}
PROPERTY MoverAccAtExit : MC_LREAL //[mm/s² on Track] Every mover that leaves or passes the station gets this new acceleration as a target.
GET
END_GET
SET
END_SET
END_PROPERTY

{attribute 'monitoring':='call'}
PROPERTY MoverDecAtExit : MC_LREAL //[mm/s² on Track] Every mover that leaves or passes the station gets this new deceleration as a target.
GET
END_GET
SET
END_SET
END_PROPERTY

{attribute 'monitoring':='call'}
PROPERTY MoverGapAtExit : LREAL //[mm] Every mover that leaves or passes the station gets this new gap as a target.
GET
END_GET
SET
END_SET
END_PROPERTY

{attribute 'monitoring':='call'}
PROPERTY MoverQueueSize : UINT
GET
END_GET
SET
END_SET
END_PROPERTY

{attribute 'monitoring':='call'}
PROPERTY MoversInPlace : BOOL
GET
END_GET
END_PROPERTY

{attribute 'monitoring':='call'}
PROPERTY MoversInQueue : REFERENCE TO ARRAY [0..(CHALET_BaseComponents.BaseParameterlist.MAX_OBJECTS-1)] OF I_XP_Mover_PLC // Return a sorted list of movers in this zone. Index 0 is the mover in Front
GET
END_GET
END_PROPERTY

{attribute 'monitoring':='call'}
PROPERTY MoverVelocityAtExit : MC_LREAL //[mm/s on Track] Every mover that leaves or passes the station gets this new velocity as a target.
GET
END_GET
SET
END_SET
END_PROPERTY

{attribute 'monitoring':='call'}
//[mm] from the beginning of the assigned track
PROPERTY PositionOnTrack : LREAL
GET
END_GET
END_PROPERTY

{attribute 'monitoring':='call'}
//Position on the assigned track
PROPERTY PositionOnTrackXY : REFERENCE TO PositionXY
GET
END_GET
END_PROPERTY

{attribute 'monitoring':='call'}
//Planned position, not necessarily on the track
PROPERTY PositionXY : REFERENCE TO  PositionXY
GET
END_GET
END_PROPERTY

{attribute 'monitoring':='call'}
PROPERTY ProcessSimulationActive : BOOL
GET
END_GET
END_PROPERTY

//The movers currently in this station must leave the station. 
//The movers actively search for a destination, but only leave if a new destination is available.
METHOD PushMoversOutOfStation : HRESULT
VAR_INPUT
END_VAR
END_METHOD

{attribute 'monitoring':='call'}
//prevent further movers from entering the station, 
//e.g. to prevent a collision. All movers that are already moving to reach this station will be stopped with a stop 
//and restarted with Ready True.
PROPERTY ReadyToRecvMovers : BOOL
GET
END_GET
SET
END_SET
END_PROPERTY

METHOD SendMoversToStation : I_CH_Feedback //All movers in the station are sent to this destination
VAR_INPUT
	sTargetStation: STRING;//unique station name or group of stations
END_VAR
END_METHOD

//If a valid time (>0seconds) is set and the configured destination station exists, then the movers will be sent away automatically after this time from now on.
METHOD SimulationStart : HRESULT
VAR_INPUT
	fProcessDuration 		: LREAL; //[s]
	sTargetStation	: STRING; //Group of the target station to automatic send after the duration
END_VAR
END_METHOD

//If a valid time (>0seconds) is set and the configured destination station exists, then the movers will be sent away automatically after this time from now on.
METHOD SimulationStartEx : HRESULT
VAR_INPUT
	fProcessDuration 		: LREAL; //[s]
	ipStation				: I_XP_Station_PLC; //unique station to automatic send after the duration
END_VAR
END_METHOD

METHOD SimulationStop : HRESULT
END_METHOD

{attribute 'monitoring':='call'}
//List of stations before this station
PROPERTY StationsAhead : I_CH_List
GET
END_GET
END_PROPERTY

{attribute 'monitoring':='call'}
//List of stations behinde this station
PROPERTY StationsBehinde : I_CH_List
GET
END_GET
END_PROPERTY

{attribute 'monitoring':='call'}
//Suppress to change the dynamic(Gap+velocity) of passing movers. This is usefull in startup
PROPERTY SuppressDynamicsChange : BOOL
GET
END_GET
SET
END_SET
END_PROPERTY

{attribute 'monitoring':='call'}
//Interface to CHALET system to which this object belongs
PROPERTY System : I_XP_System_PLC
GET
END_GET
END_PROPERTY

{attribute 'monitoring':='call'}
PROPERTY TargetGroupe : STRING
GET
END_GET
END_PROPERTY

{attribute 'monitoring':='call'}
//A time that is waited as soon as the mover is in the station (including the monitoring window) before “MoversInPlace” is set. e.g. used to stabilize the workpiece
PROPERTY TargetPosMonitoringTime : TIME
GET
END_GET
SET
END_SET
END_PROPERTY

{attribute 'monitoring':='call'}
//How many mm before the mover reaches the position is “MoversInPlace” set for the process. 
//This distance can also be set very large (e.g. 100mm) for moving past without stopping.
PROPERTY TargetPosWindow : LREAL
GET
END_GET
SET
END_SET
END_PROPERTY

END_INTERFACE

// ---- COMPONENTs/Environment/I_XP_Environment.TcIO
INTERFACE I_XP_Environment EXTENDS I_CH_Object

METHOD AddToGroup : HRESULT
VAR_INPUT
	iGroup : I_XP_Group;
END_VAR
END_METHOD

(* Clears the Planar Environment (stators and boundary). *)
METHOD Clear : HRESULT
END_METHOD

METHOD Configure : HRESULT
VAR_INPUT
END_VAR
END_METHOD

{attribute 'monitoring':='call'}
PROPERTY Feedback : I_XP_Feedback
GET
END_GET
END_PROPERTY

METHOD Initialize : HRESULT
END_METHOD

{attribute 'monitoring':='call'}
PROPERTY Mapped : BOOL //Project is mapped to MC (McToPlc and PlcToMc)
GET
END_GET
END_PROPERTY

{attribute 'monitoring':='call'}
//Unique object ID
PROPERTY OID : OTCID
GET
END_GET
END_PROPERTY

{attribute 'monitoring':='call'}
PROPERTY PlanarEnvironment : REFERENCE TO MC_PlanarEnvironment
GET
END_GET
END_PROPERTY

{attribute 'monitoring':='call'}
//Enumeration MoverDetectionStatus
PROPERTY ProcessingUnitMoverDetectionStatus : MoverDetectionStatus
GET
END_GET
END_PROPERTY

{attribute 'monitoring':='call'}
//Object ID of the IoXPlanar processing unit
PROPERTY ProcessingUnitOID : OTCID
GET
END_GET
END_PROPERTY

METHOD RemoveFromGroup : HRESULT
END_METHOD

METHOD PUBLIC Update : HRESULT
VAR_INPUT
END_VAR
END_METHOD

{attribute 'monitoring':='call'}
PROPERTY UtilityEnvirement : Tc3_XPlanarUtility.I_Environment
GET
END_GET
END_PROPERTY

END_INTERFACE

// ---- COMPONENTs/Group/I_XP_Group.TcIO
INTERFACE I_XP_Group  EXTENDS I_CH_Object

METHOD AddEnvironment : HRESULT
VAR_INPUT
	refEnvironment : REFERENCE TO MC_PlanarEnvironment;
	refFeedback : REFERENCE TO MC_PlanarFeedback;
END_VAR
END_METHOD

METHOD AddMover : HRESULT
VAR_INPUT
	refMover : REFERENCE TO MC_PlanarMover;
	refFeedback : REFERENCE TO MC_PlanarFeedback;
END_VAR
END_METHOD

METHOD AddTrack : HRESULT
VAR_INPUT
	refTrack : REFERENCE TO MC_PlanarTrack;
	refFeedback : REFERENCE TO MC_PlanarFeedback;
END_VAR
END_METHOD

METHOD Disable : HRESULT
VAR_INPUT
END_VAR
END_METHOD

METHOD Enable : HRESULT
VAR_INPUT
END_VAR
END_METHOD

{attribute 'OPC.UA.DA.Property' := '1'}
{attribute 'monitoring':='call'}
PROPERTY Feedback : I_XP_Feedback
GET
END_GET
END_PROPERTY

METHOD Initialize : HRESULT
VAR_INPUT
END_VAR
END_METHOD

{attribute 'monitoring':='call'}
PROPERTY Mapped : BOOL //Project is mapped to MC (McToPlc and PlcToMc)
GET
END_GET
END_PROPERTY

{attribute 'monitoring':='call'}
//Unique object ID
PROPERTY OID : OTCID
GET
END_GET
END_PROPERTY

{attribute 'monitoring':='call'}
PROPERTY PlanarGroup : REFERENCE TO MC_PlanarGroup
GET
END_GET
END_PROPERTY

METHOD Reset : HRESULT
VAR_INPUT
END_VAR
END_METHOD

METHOD PUBLIC Update : HRESULT
VAR_INPUT
END_VAR
END_METHOD

END_INTERFACE

// ---- COMPONENTs/System/I_XP_System_PLC.TcIO
INTERFACE I_XP_System_PLC EXTENDS I_CH_Object

METHOD CheckTargetExists : BOOL //Return TRUE if target is existing
VAR_INPUT
	sStation	: STRING; //Group of the target station or LUID
END_VAR
END_METHOD

METHOD Disable : I_CH_Feedback
VAR_INPUT
END_VAR
END_METHOD

{attribute 'monitoring':='call'}
PROPERTY Disabled : BOOL
GET
END_GET
END_PROPERTY

METHOD Enable : I_CH_Feedback
VAR_INPUT
END_VAR
END_METHOD

{attribute 'monitoring':='call'}
PROPERTY Enabled : BOOL
GET
END_GET
END_PROPERTY

{attribute 'monitoring':='call'}
PROPERTY Enviroment : I_XP_Environment
GET
END_GET
END_PROPERTY

METHOD FastStop : I_CH_Feedback
END_METHOD

{attribute 'monitoring':='call'}
PROPERTY Feedback : CHALET_BaseComponents.I_CH_Feedback
GET
END_GET
END_PROPERTY

//Returns the station that is closest to the point according to Phytagoras
METHOD GetStationClosestTo : I_XP_Station
VAR_INPUT
	pos : MoverVector;
END_VAR
END_METHOD

METHOD Initialize : HRESULT
VAR_INPUT
END_VAR
END_METHOD

{attribute 'monitoring':='call'}
PROPERTY Initialized : BOOL
GET
END_GET
END_PROPERTY

{attribute 'monitoring':='call'}
//List of movers that are not present in the current system
PROPERTY MoversNotPresent : CHALET_BaseComponents.I_CH_LIST
GET
END_GET
END_PROPERTY

{attribute 'monitoring':='call'}
//List of movers that are present in the current system
PROPERTY MoversPresent : CHALET_BaseComponents.I_CH_LIST
GET
END_GET
END_PROPERTY

{attribute 'monitoring':='call'}
PROPERTY Paths : CHALET_BaseComponents.I_CH_LIST
GET
END_GET
END_PROPERTY

METHOD Station : I_XP_Station_PLC
VAR_INPUT
	sLUID : STRING;
END_VAR
END_METHOD

{attribute 'monitoring':='call'}
//List of all station objects that exist in this project
PROPERTY StationsAll : CHALET_BaseComponents.I_CH_LIST
GET
END_GET
END_PROPERTY

{attribute 'monitoring':='call'}
//List of all station objects that are considered for path planning in the currently running system
PROPERTY StationsUsed : CHALET_BaseComponents.I_CH_LIST
GET
END_GET
END_PROPERTY

//Suppress to change the dynamic(Gap) of passing movers in all stations. This is usefull in startup
PROPERTY SuppressAllDynamicsChanges : BOOL
SET
END_SET
END_PROPERTY

{attribute 'monitoring':='call'}
PROPERTY Tracks : CHALET_BaseComponents.I_CH_LIST
GET
END_GET
END_PROPERTY

{attribute 'monitoring':='call'}
PROPERTY Triggers : CHALET_BaseComponents.I_CH_LIST
GET
END_GET
END_PROPERTY

METHOD Update : HRESULT
VAR_INPUT
END_VAR
END_METHOD

{attribute 'monitoring':='call'}
PROPERTY Zones : CHALET_BaseComponents.I_CH_LIST
GET
END_GET
END_PROPERTY

END_INTERFACE

// ---- COMPONENTs/System/I_XP_System_Registration.TcIO
INTERFACE I_XP_System_Registration EXTENDS __SYSTEM.IQueryInterface

{attribute 'monitoring':='call'}
PROPERTY Disabled : BOOL
GET
END_GET
END_PROPERTY

{attribute 'monitoring':='call'}
PROPERTY Enabled : BOOL
GET
END_GET
END_PROPERTY

{attribute 'monitoring':='call'}
PROPERTY Enviroment : I_XP_Environment
GET
END_GET
END_PROPERTY

METHOD LinkEnvironment : HRESULT
VAR_INPUT
	ipEnvironment : I_CH_Object;
END_VAR
END_METHOD

METHOD LinkGroup : HRESULT
VAR_INPUT
	ipGroup : I_CH_Object;
END_VAR
END_METHOD

{attribute 'monitoring':='call'}
//List of movers that are not present in the current system
PROPERTY MoversNotPresent : CHALET_BaseComponents.I_CH_LIST
GET
END_GET
END_PROPERTY

{attribute 'monitoring':='call'}
//List of movers that are present in the current system
PROPERTY MoversPresent : CHALET_BaseComponents.I_CH_LIST
GET
END_GET
END_PROPERTY

{attribute 'monitoring':='call'}
PROPERTY Paths : CHALET_BaseComponents.I_CH_LIST
GET
END_GET
END_PROPERTY

METHOD RegisterMover : HRESULT
VAR_INPUT
	ipMover : I_CH_Object;
END_VAR
END_METHOD

METHOD RegisterStation : HRESULT
VAR_INPUT
	ipStation : I_CH_Object;
END_VAR
END_METHOD

METHOD RegisterTrack : HRESULT
VAR_INPUT
	ipTrack : I_CH_Object;
END_VAR
END_METHOD

METHOD RegisterTrigger : HRESULT
VAR_INPUT
	ipTrigger	: CHALET_BaseComponents.I_CH_Object;
END_VAR
END_METHOD

METHOD RegisterZone : HRESULT
VAR_INPUT
	ipZone	: CHALET_BaseComponents.I_CH_Object;
END_VAR
END_METHOD

{attribute 'monitoring':='call'}
//List of all station objects that exist in this project
PROPERTY StationsAll : CHALET_BaseComponents.I_CH_LIST
GET
END_GET
END_PROPERTY

{attribute 'monitoring':='call'}
//List of all station objects that are considered for path planning in the currently running system
PROPERTY StationsUsed : CHALET_BaseComponents.I_CH_LIST
GET
END_GET
END_PROPERTY

{attribute 'monitoring':='call'}
PROPERTY Tracks : CHALET_BaseComponents.I_CH_LIST
GET
END_GET
END_PROPERTY

{attribute 'monitoring':='call'}
PROPERTY Triggers : CHALET_BaseComponents.I_CH_LIST
GET
END_GET
END_PROPERTY

{attribute 'monitoring':='call'}
PROPERTY Zones : CHALET_BaseComponents.I_CH_LIST
GET
END_GET
END_PROPERTY

END_INTERFACE

// ---- COMPONENTs/Track/I_XP_Track.TcIO
INTERFACE I_XP_Track  EXTENDS I_CH_Object

METHOD AddMover : HRESULT
VAR_INPUT
	ipMover : I_XP_Mover;
END_VAR
END_METHOD

METHOD AddToGroup : HRESULT
VAR_INPUT
	iGroup : I_XP_Group;
END_VAR
END_METHOD

{attribute 'monitoring':='call'}
PROPERTY ClosedLoop : BOOL
GET
END_GET
END_PROPERTY

METHOD Configure : HRESULT
VAR_INPUT
END_VAR
END_METHOD

METHOD Configuring : HRESULT
VAR_INPUT
END_VAR
END_METHOD

{attribute 'monitoring':='call'}
PROPERTY CtsMoversOnTrack : UINT
GET
END_GET
END_PROPERTY

METHOD Disable : HRESULT
VAR_INPUT
END_VAR
END_METHOD

METHOD Enable : HRESULT
VAR_INPUT
END_VAR
END_METHOD

{attribute 'monitoring':='call'}
//Position of the end point of this tracks
PROPERTY EndPosition : REFERENCE TO MoverVector
GET
END_GET
END_PROPERTY

{attribute 'monitoring':='call'}
PROPERTY Feedback : I_XP_Feedback
GET
END_GET
END_PROPERTY

(* Calculates which gap the mover should have on a position
	The gap results from the last station crossed.
	If several stations are possible ( switch), the largest gap is displayed here *)
METHOD GapAtPosition : LREAL
VAR_INPUT
	fPosOnTrack : LREAL;//[mm]	
END_VAR
END_METHOD

//Each track has an auxiliary station at the end of itself. This is used automatically or not, depending on whether the track also contains stations created by the user.
//These are used by the movers as auxiliary links to navigate through a complex network.
{attribute 'monitoring':='call'}
PROPERTY HelperStationAtEndOfTrack : I_XP_Station
GET
END_GET
END_PROPERTY

{attribute 'monitoring':='call'}
//[mm]
PROPERTY Length : LREAL
GET
END_GET
END_PROPERTY

{attribute 'monitoring':='call'}
PROPERTY PlanarTrack : REFERENCE TO MC_PlanarTrack
GET
END_GET
END_PROPERTY

METHOD RemoveFromGroup : HRESULT
END_METHOD

METHOD Reset : HRESULT
VAR_INPUT
END_VAR
END_METHOD

{attribute 'monitoring':='call'}
//Position of the start point of this tracks
PROPERTY StartPosition : REFERENCE TO MoverVector
GET
END_GET
END_PROPERTY

(* Returns the first station on current track who has exact thsi position or is ahead
	If no station on this track, result is maybe on another track*)
METHOD StationAhedPosition : I_XP_Station
VAR_INPUT
	fPosOnTrack : LREAL;//[mm]	
END_VAR
END_METHOD

(* Returns the first station on current track who has exact this position or is behind
	If no station on this track, result is maybe on another track*)
METHOD StationBehindPosition : I_XP_Station
VAR_INPUT
	fPosOnTrack : LREAL;//[mm]	
END_VAR
END_METHOD

(* Returns the closest station on current, ahead or behind track*)
METHOD StationClosestTo : I_XP_Station
VAR_INPUT
	fPosOnTrack : LREAL;//[mm]	
END_VAR
END_METHOD

{attribute 'monitoring':='call'}
//List of interfaces to stations on this track
PROPERTY StationsOnTrack : I_CH_List
GET
END_GET
END_PROPERTY

{attribute 'monitoring':='call'}
//List of interfaces from other tracks
PROPERTY TracksAhead : I_CH_List
GET
END_GET
END_PROPERTY

{attribute 'monitoring':='call'}
//List of interfaces from other tracks
PROPERTY TracksBehinde : I_CH_List
GET
END_GET
END_PROPERTY

{attribute 'monitoring':='call'}
PROPERTY TracksEndAtThis : REFERENCE TO  ARRAY[0..(XPlanarParameterlist.N_MAX_STATIONS_AHEAD_OR_BEHIND-1)] OF I_XP_Track
GET
END_GET
END_PROPERTY

{attribute 'monitoring':='call'}
PROPERTY TracksStartFromThis : REFERENCE TO ARRAY[0..(XPlanarParameterlist.N_MAX_STATIONS_AHEAD_OR_BEHIND-1)] OF I_XP_Track
GET
END_GET
END_PROPERTY

{attribute 'monitoring':='call'}
//Interface to this track in XPlanar Utility Lib
PROPERTY UtilityTrack : Tc3_XPlanarUtility.I_McPlanarTrack
GET
END_GET
END_PROPERTY

END_INTERFACE

// ---- COMPONENTs/Track/I_XP_Track_PLC.TcIO
INTERFACE I_XP_Track_PLC EXTENDS I_CH_Object

{attribute 'monitoring':='call'}
PROPERTY CtsMoversOnTrack : UINT
GET
END_GET
END_PROPERTY

{attribute 'monitoring':='call'}
//Position of the end point of this tracks
PROPERTY EndPosition : REFERENCE TO MoverVector
GET
END_GET
END_PROPERTY

{attribute 'monitoring':='call'}
PROPERTY Feedback : I_XP_Feedback
GET
END_GET
END_PROPERTY

{attribute 'monitoring':='call'}
//[mm]
PROPERTY Length : LREAL
GET
END_GET
END_PROPERTY

{attribute 'monitoring':='call'}
PROPERTY Mapped : BOOL //Project is mapped to MC (McToPlc and PlcToMc)
GET
END_GET
END_PROPERTY

{attribute 'monitoring':='call'}
// Number of elements describing the geometric curve of the track.
PROPERTY NbOfGeometricElements : UINT
GET
END_GET
END_PROPERTY

{attribute 'monitoring':='call'}
//Unique object ID
PROPERTY OID : OTCID
GET
END_GET
END_PROPERTY

{attribute 'monitoring':='call'}
PROPERTY PlanarTrack : REFERENCE TO MC_PlanarTrack
GET
END_GET
END_PROPERTY

//The geometric points of a track are copied. Including the position and type. This only works if the system is disabled.
METHOD ReplicateGeometricElements : HRESULT
VAR_INPUT
	ipTrackCopyFrom : I_XP_Track;
END_VAR
END_METHOD

//move all points of the track geometry. Only works if the system is disabled.
METHOD ShiftTrack : HRESULT
VAR_INPUT
	xOffset, yOffset : LREAL;
END_VAR
END_METHOD

{attribute 'monitoring':='call'}
//Position of the start point of this tracks
PROPERTY StartPosition : REFERENCE TO MoverVector
GET
END_GET
END_PROPERTY

(* Returns the first station on current track who has exact thsi position or is ahead
	If no station on this track, result is maybe on another track*)
METHOD StationAhedPosition : I_XP_Station
VAR_INPUT
	fPosOnTrack : LREAL;//[mm]	
END_VAR
END_METHOD

(* Returns the first station on current track who has exact thsi position or is behind
	If no station on this track, result is maybe on another track*)
METHOD StationBehindPosition : I_XP_Station
VAR_INPUT
	fPosOnTrack : LREAL;//[mm]	
END_VAR
END_METHOD

(* Returns the closest station on current, ahead or behind track*)
METHOD StationClosestTo : I_XP_Station
VAR_INPUT
	fPosOnTrack : LREAL;//[mm]	
END_VAR
END_METHOD

{attribute 'monitoring':='call'}
//List of interfaces to stations on this track
PROPERTY StationsOnTrack : I_CH_List
GET
END_GET
END_PROPERTY

{attribute 'monitoring':='call'}
//Interface to CHALET system to which this object belongs
PROPERTY System : I_XP_System_PLC
GET
END_GET
END_PROPERTY

{attribute 'monitoring':='call'}
//List of interfaces from other tracks
PROPERTY TracksAhead : I_CH_List
GET
END_GET
END_PROPERTY

{attribute 'monitoring':='call'}
//List of interfaces from other tracks
PROPERTY TracksBehinde : I_CH_List
GET
END_GET
END_PROPERTY

{attribute 'monitoring':='call'}
PROPERTY TracksEndAtThis : REFERENCE TO  ARRAY[0..(XPlanarParameterlist.N_MAX_STATIONS_AHEAD_OR_BEHIND-1)] OF I_XP_Track
GET
END_GET
END_PROPERTY

{attribute 'monitoring':='call'}
PROPERTY TracksStartFromThis : REFERENCE TO ARRAY[0..(XPlanarParameterlist.N_MAX_STATIONS_AHEAD_OR_BEHIND-1)] OF I_XP_Track
GET
END_GET
END_PROPERTY

{attribute 'monitoring':='call'}
//Interface to this track in XPlanar Utility Lib
PROPERTY UtilityTrack : Tc3_XPlanarUtility.I_McPlanarTrack
GET
END_GET
END_PROPERTY

END_INTERFACE

// ---- COMPONENTs/Feedback/FB_XP_Feedback.TcPOU
{attribute 'no_explicit_call' := 'Do not call the body - Stick to OOP'}
FUNCTION_BLOCK FB_XP_Feedback EXTENDS CHALET_Nc.FB_NcFeedback IMPLEMENTS I_XP_Feedback
VAR_INPUT
END_VAR
VAR_OUTPUT
END_VAR
VAR
	(* Indicates which object one would collide with. *)
	{attribute 'hide'}
	_objectInfo : ST_PlanarObjectInfoEx;
END_VAR

METHOD ClearObjectInfo : BOOL
VAR_INPUT
END_VAR
THIS^._ObjectInfo.Id := 0;
THIS^._ObjectInfo.ipObject := 0;
THIS^._ObjectInfo.ObjectType := EPlanarObjectType.None;
END_METHOD

{attribute 'monitoring':='call'}
(* Indicates which object one would collide with. *)
PROPERTY ObjectInfo : REFERENCE TO PlanarObjectInfo
GET
objectInfo REF= THIS^._objectInfo;
END_GET
SET
THIS^._objectInfo.Id			:= ObjectInfo.Id;
THIS^._objectInfo.ObjectType 	:= ObjectInfo.ObjectType;
THIS^._objectInfo.ipObject 		:= 0;
END_SET
END_PROPERTY

{attribute 'monitoring':='call'}
(* Indicates which object one would collide with. *)
PROPERTY ObjectInfoEx : REFERENCE TO ST_PlanarObjectInfoEx
GET
objectInfoEx REF= THIS^._objectInfo;
END_GET
SET
THIS^._objectInfo := ObjectInfoEx;
END_SET
END_PROPERTY

END_FUNCTION_BLOCK

// ---- COMPONENTs/Mover/FB_XP_Mover.TcPOU
// The warning " Interface of overridden methode xxx of base I_xxx doesn't match declaration" can be disabled here. 
{warning disable C0094 }
{attribute 'no_explicit_call' := 'Do not call the body - Stick to OOP'}
(* XPlanar mover - n per associated XPlanar. Can be instantiated as an array and/or individually
	The Planar mover is a software object that represents an XPlanar mover. It summarizes the state of the real mover (position, velocity, etc.) 
	for the user. In addition, the user has the possibility to influence or control the state of the real mover via the Planar mover. *)	
FUNCTION_BLOCK FB_XP_Mover EXTENDS FB_CH_Object IMPLEMENTS I_XP_Mover, I_XP_Mover_PLC
VAR
	fbRouteRemaining : FB_CH_List;//Remaining route to the parent station
	fbRouteComplete : FB_CH_List;//Complete route from last parent to active parent station
END_VAR

VAR
	//Link to MC-Mover
	fbMover : MC_PlanarMover; 
	
	{attribute 'hide'}  
	bInitDone :BOOL := FALSE;
	{attribute 'hide'}               	
	fbFeedback 			: FB_XP_Feedback(ipSourceInfo := fbSourceInfo);	
	{attribute 'hide'}                   	
	eActiveCommand 		: CHALET_Nc.E_NcAxisCommands := CHALET_Nc.E_NcAxisCommands.None;
	{attribute 'hide'}
	ipXpSystem : I_XP_System_Registration;
	{attribute 'hide'} 
	sTargetStation : STRING := XPlanarParameterlist.S_MOVER_TARGED_INIT;
	{attribute 'hide'} 
	sCurrentStation : STRING;
	{attribute 'hide'}
	ipParentStation : I_XP_Station; //This is the station in which the Mover is currently standing or moving.	
	{attribute 'hide'}
	ipProductData : I_XP_ProductData; //later the required interface of the tool or product can be queried via query interface
	{attribute 'hide'}	
	ipMcMover : Tc3_XPlanarUtility.I_McPlanarMover;
	{attribute 'hide'}	
	ipTcIoMover : Tc3_XPlanarUtility.I_TcIoXPlanarMover;
END_VAR

//Recovery
VAR
	{attribute 'hide'}
	stLastValidPositionXYZABC :  MoverVector;//This was the last valid (system enabled) actual  position of the mover
	{attribute 'hide'}
	//This was the last valid (system enabled) actual  position of the mover
	fLastValidPositionOnTrack :  LREAL;
	{attribute 'hide'}
	ipLastValidTrack : I_XP_Track;	//This was the last valid (system enabled) actual  position of the mover
	{attribute 'hide'}
	fLastCmdTargetPosition : LREAL; //the last commanded target position [mm]
	{attribute 'hide'}	
	fLastCmdTargetGap 	: LREAL; //the last commanded target gap
	{attribute 'hide'}		
	ipLastCmdTrack : I_XP_Track; //the last commanded target track
	{attribute 'hide'}			
	ipLastValidParentStation : I_XP_Station; //the last commanded parent station
END_VAR


//External Setpoint Generator
VAR
	AxisSetpointX : FB_NcAxis;
	AxisSetpointY : FB_NcAxis;
	AxisSetpointZ : FB_NcAxis;
	AxisSetpointA : FB_NcAxis;
	AxisSetpointB : FB_NcAxis;
	AxisSetpointC : FB_NcAxis;
	{attribute 'hide'} 
	nSeqStartExternalSetpoint : UINT;
	{attribute 'hide'} 	
	//As long as the bit is still false, the MC_PlanarFeedback should not be evaluated as it may still indicate an old error
	bEvaluateFeedback: BOOL; 
	{attribute 'hide'} 
	bFeedExternalSetpointActive : BOOL; 
	{attribute 'hide'} 
	fbFeedbackExternalSetpointStartSeq : FB_CH_Feedback(0);
	{attribute 'hide'} 
	ipMasterMover : I_XP_Mover;	
	{attribute 'hide'} 
	stMasterMovementScaling : MoverVector; // if 0, Mover is not folowing this mover axis
	{attribute 'hide'} 
	stMasterPositionAtStart : MoverVector;
END_VAR


//Unknown Level
VAR
//	{attribute 'hide'} 
	nSeqLiftFromUnknown : UINT;
//	{attribute 'hide'} 
	nSeqLowerToUnknown : UINT;	
//	{attribute 'hide'} 
	fbFeedbackLiftFromUnknown  : FB_CH_Feedback(0);
//	{attribute 'hide'} 
	fbFeedbackLowerToUnknown : FB_CH_Feedback(0);
END_VAR


//DynamicConstraint
VAR
	{attribute 'hide'} 
	fbDynConstraintContainer 	: DynamicConstraint_Container;		//A container for dynamic constraints.
	{attribute 'hide'} 
	fbDynConstraintPath 		: DynamicConstraint_PathXY; 		//One dimensional dynamic constraint along the XY-components of a path, ignoring non-tangential effects.
	{attribute 'hide'} 	
	fbDynConstraintCoordinates	: DynamicConstraint_Coordinates;	//Dynamic constraints for individual coordinates.
END_VAR


// Planar-Feedback objects
VAR
	{attribute 'hide'} 
	fbFeedbackMoveA : MC_PlanarFeedback;
	{attribute 'hide'} 
	fbFeedbackMoveB : MC_PlanarFeedback;
	{attribute 'hide'} 
	fbFeedbackMoveC : MC_PlanarFeedback;
	{attribute 'hide'} 
	fbFeedbackMoveXY : MC_PlanarFeedback;
	{attribute 'hide'} 
	fbFeedbackMoveZ : MC_PlanarFeedback;
	{attribute 'hide'} 
	fbFeedbackEnable : MC_PlanarFeedback;
	{attribute 'hide'} 
	fbFeedbackDisable : MC_PlanarFeedback;
	{attribute 'hide'} 
	fbFeedbackHalt : MC_PlanarFeedback;
	{attribute 'hide'} 
	fbFeedbackReset : MC_PlanarFeedback;
	{attribute 'hide'} 
	fbFeedbackAddToGrp : MC_PlanarFeedback;
	{attribute 'hide'} 
	fbFeedbackRmvFromGrp : MC_PlanarFeedback;
	{attribute 'hide'} 
	fbFeedbackJoinTrack : MC_PlanarFeedback;
	{attribute 'hide'} 
	fbFeedbackMoveOnTrack: MC_PlanarFeedback;	
	{attribute 'hide'} 
	fbFeedbackExtStart : MC_PlanarFeedback;
	{attribute 'hide'} 
	fbFeedbackExtStop : MC_PlanarFeedback;
END_VAR
{warning restore C0094}

{attribute 'monitoring':='call'}
(* Provides the current planar mover setpoint XYZABC [mm/s²] *)
PROPERTY AccelerationSet : REFERENCE TO MoverVector
GET
VAR_INST
	{attribute 'hide'}
	copyOfData :  MoverVector;
END_VAR
//Creat an copy of the struct to view value in targetdbrowser and plc online view
copyOfData := THIS^.fbMover.MCTOPLC.SET.SetAcc;
AccelerationSet REF= copyOfData;
END_GET
END_PROPERTY

//Save the master mover and apply the distance traveled as a relative offset to this slave mover. Requires .StartExternalSetpoint()
METHOD AddMoverExtSetpoint : HRESULT
VAR_INPUT
	ipMasterMover : I_XP_Mover;
	fScalingX, fScalingY, fScalingZ, fScalingA, fScalingB, fScalingC : LREAL;// If >0, follow this axis to master-mover
END_VAR
//Invalide input
IF ipMasterMover = 0 THEN
	AddMoverExtSetpoint := E_FAIL;
	RETURN;
END_IF

//Allready stored a master
IF THIS^.ipMasterMover <> 0 THEN
	AddMoverExtSetpoint := E_FAIL;
	RETURN;
END_IF

//Only possible if ExternalSetpoint is not running
IF THIS^.nSeqStartExternalSetpoint <> 0 THEN
	AddMoverExtSetpoint := E_FAIL;
	RETURN;
END_IF



THIS^.ipMasterMover := ipMasterMover;
THIS^.stMasterMovementScaling.x := fScalingX;
THIS^.stMasterMovementScaling.y := fScalingy;
THIS^.stMasterMovementScaling.z := fScalingz;
THIS^.stMasterMovementScaling.a := fScalinga;
THIS^.stMasterMovementScaling.b := fScalingb;
THIS^.stMasterMovementScaling.c := fScalingc;
END_METHOD

METHOD AddToGroup : HRESULT
VAR_INPUT
	iGroup : I_XP_Group;
END_VAR
IF NOT THIS^.fbFeedback.Busy THEN
	THIS^.eActiveCommand 				:= CHALET_NC.E_NcAxisCommands.AddToGroupe;
	THIS^.fbFeedback.ActiveCommand 		:= TO_STRING(THIS^.eActiveCommand);	
	THIS^.fbFeedback.LastCommandAccepted:= TRUE;		
	THIS^.fbFeedback.Busy 				:= TRUE;
	
	iGroup.AddMover(THIS^.fbMover, THIS^.fbFeedbackAddToGrp);
	AddToGroup := S_OK;
ELSE
	AddToGroup := S_FALSE;
	THIS^.fbFeedback.LastCommandAccepted:= FALSE;	
END_IF
END_METHOD

{attribute 'monitoring':='call'}
PROPERTY  AxisExtSetpointA : CHALET_Nc.I_NcAxis_PLC
GET
AxisExtSetpointA := THIS^.AxisSetpointA;
END_GET
END_PROPERTY

{attribute 'monitoring':='call'}
PROPERTY AxisExtSetpointB : CHALET_Nc.I_NcAxis_PLC
GET
AxisExtSetpointB := THIS^.AxisSetpointB;
END_GET
END_PROPERTY

{attribute 'monitoring':='call'}
PROPERTY AxisExtSetpointC : CHALET_Nc.I_NcAxis_PLC
GET
AxisExtSetpointC := THIS^.AxisSetpointC;
END_GET
END_PROPERTY

{attribute 'monitoring':='call'}
PROPERTY  AxisExtSetpointX : CHALET_Nc.I_NcAxis_PLC
GET
AxisExtSetpointX := THIS^.AxisSetpointX;
END_GET
END_PROPERTY

{attribute 'monitoring':='call'}
PROPERTY AxisExtSetpointY : CHALET_Nc.I_NcAxis_PLC
GET
AxisExtSetpointY := THIS^.AxisSetpointY;
END_GET
END_PROPERTY

{attribute 'monitoring':='call'}
PROPERTY AxisExtSetpointZ : CHALET_Nc.I_NcAxis_PLC
GET
AxisExtSetpointZ := THIS^.AxisSetpointZ;
END_GET
END_PROPERTY

{attribute 'monitoring':='call'}
(* C coordinate modulus set in MC3-Planar Mover[°] *)
PROPERTY CAxisModulo : LREAL
GET
VAR
	ipTrackComObject : ITComObject;
	nParaSize : UDINT;
	pParaData : PVOID;
	hr : HRESULT;
	fData : LREAL;
END_VAR
VAR CONSTANT
	N_IDX_OFFSET 	: UDINT := 16#05030107; // Parameter(init) Mover
END_VAR
FW_ObjMgr_GetObjectInstance(oid:= THIS^.OID, iid:= TC_GLOBAL_IID_LIST.IID_ITComObject, pipUnk:= ADR(ipTrackComObject));

IF ipTrackComObject = 0 THEN
	// Error
	RETURN;
END_IF


nParaSize := SIZEOF(fData);	pParaData := ADR(fData);

hr := ipTrackComObject.TcGetObjPara(pid:=N_IDX_OFFSET , nData:= nParaSize, pData:= pParaData, pgp:=0 );
FW_SafeRelease(ADR(ipTrackComObject));


CAxisModulo := TO_LREAL(TO_DINT(fData));
END_GET
END_PROPERTY

{attribute 'monitoring':='call'}
(* Indicates the command mode of an enabled PlanarMover, i.e. how setpoints are currently produced. *)
PROPERTY CommandMode : MC_PLANAR_MOVER_COMMAND_MODE
GET
CommandMode := THIS^.fbMover.MCTOPLC.STD.CommandMode;
END_GET
END_PROPERTY

{attribute 'monitoring':='call'}
PROPERTY CurrentTrack : I_XP_Track
GET
VAR
	ipTrackObj : I_CH_Object;
	ipTrack : I_XP_Track;
END_VAR
IF ipXpSystem <> 0 THEN
	ipTrackObj := ipXpSystem.Tracks.FindOID(THIS^.PlanarMover.MCTOPLC.SETONTRACK.TrackOID);
	ToXpTrack(ipTrackObj,ipTrack);
END_IF

CurrentTrack := ipTrack;
END_GET
END_PROPERTY

METHOD Disable : HRESULT
VAR_INPUT
END_VAR
THIS^.eActiveCommand 				:= CHALET_NC.E_NcAxisCommands.Disable;
THIS^.fbFeedback.ActiveCommand 		:= TO_STRING(THIS^.eActiveCommand);	
THIS^.fbFeedback.LastCommandAccepted:= TRUE;		
THIS^.fbFeedback.Busy 				:= TRUE;

//Disable Axis
THIS^.fbMover.Disable(THIS^.fbFeedbackDisable);
Disable := S_OK;
END_METHOD

//This method is called when the system is disabled. Links are deleted as they may no longer be valid
METHOD Disassemble : HRESULT
VAR_INPUT
END_VAR

//Todo zzz Braucht es diese methode noch?
fbRouteComplete.Clear(); 
fbRouteRemaining.Clear(); 


Disassemble := S_OK;
END_METHOD

{attribute 'monitoring':='call'}
//Distance to the responsible parent station [mm]
PROPERTY DistToParentStation : LREAL
GET
VAR
	fDistToParentStationStartup : LREAL := CHALET_BaseComponents.GVL_Datatypes.cMaxLreal;
	fDistToParentStationReturn : LREAL;
	
	
	ipPath : I_XP_Path;
	bPathFound : BOOL;
	fTempDistToDest : LREAL;
	
	refPosOnTrack : REFERENCE TO MoverVector;
	ipNextWaypoint : I_XP_Station;
	
	fTotalLength : LREAL;
	fDistToBegin : LREAL;
END_VAR
IF THIS^.ParentStation = 0 THEN
	DistToParentStation := CHALET_BaseComponents.GVL_Datatypes.cMaxLreal;
	RETURN;
END_IF

//--- Not on track, line 
IF THIS^.CurrentTrack = 0 THEN
	refPosOnTrack REF= THIS^.ParentStation.PositionOnTrackXYZABC;
	fDistToParentStationReturn := F_DistXYVectors(THIS^.PositionAct,refPosOnTrack);
// ---- ---- ----	


//--- at startup there is no route - parent is station ahead
ELSIF THIS^.fbRouteComplete.IsEmpty THEN
	//check each path behind the parentstation if the mover is on it
	ParentStation.PathsBehinde.ResetIterator();
	WHILE ParentStation.PathsBehinde.HasNextObject() DO
		IF __QUERYINTERFACE(ParentStation.PathsBehinde.GetNextObject(), ipPath) THEN
			//get shortest distance
			fDistToParentStationStartup:= MIN(ipPath.DistanceToDestiantion(ipTrack:= THIS^.CurrentTrack, fPosOnTrack := THIS^.PositionOnTrack), fDistToParentStationStartup);
		END_IF
	END_WHILE
	ParentStation.PathsBehinde.RestoreIterator();	
	fDistToParentStationReturn := fDistToParentStationStartup;
// ---- ---- ----

// ---- Normal route dureing enabled system
ELSE
	THIS^.fbRouteComplete.ResetIterator();
	WHILE THIS^.fbRouteComplete.HasNextObject() DO
		IF __QUERYINTERFACE(THIS^.fbRouteComplete.GetNextObject(), ipPath) THEN
			fTotalLength := fTotalLength + ipPath.Length;
		
			IF NOT bPathFound THEN
				fTempDistToDest := ipPath.DistanceToDestiantion(ipTrack := THIS^.CurrentTrack, fPosOnTrack := THIS^.PositionOnTrack); 
				IF 	fTempDistToDest <> CHALET_BaseComponents.GVL_Datatypes.cMaxLreal THEN
					bPathFound := TRUE;
					fDistToParentStationReturn := fTempDistToDest;
				END_IF
			ELSE 
				fDistToParentStationReturn := fDistToParentStationReturn + ipPath.Length;
			END_IF
		END_IF
	END_WHILE
	THIS^.fbRouteComplete.RestoreIterator();
	// ---- ---- ----
	
	
	//--- If Mover is not on the path, return total length + dist to beginn
	IF NOT bPathFound THEN
		THIS^.fbRouteComplete.ResetIterator();
		IF __QUERYINTERFACE(THIS^.fbRouteComplete.GetNextObject(), ipPath) THEN
			refPosOnTrack REF= ipPath.StationDestination.PositionOnTrackXYZABC;
			fDistToBegin := F_DistXYVectors(THIS^.PositionAct, refPosOnTrack);	
		END_IF
		THIS^.fbRouteComplete.RestoreIterator();
		
		
		fDistToParentStationReturn := fDistToBegin + fTotalLength;
	END_IF
	 // ---- ---- ----

END_IF
// ---- ---- ----

DistToParentStation := fDistToParentStationReturn;

//Todo absturz, maximalwert von LREAL überschritten
//redce to 3 decimal places
//DistToParentStation := DINT_TO_LREAL(LREAL_TO_DINT(fDistToParentStationReturn*1000))/1000.0;
END_GET
END_PROPERTY

METHOD DistToTrack : LREAL
VAR_INPUT
	iTrack : I_XP_Track;
END_VAR
VAR
	fPositionOnTrack : LREAL;
	trackPosition, moverPosition : PositionXYC;
END_VAR
moverPosition.x := PositionSet.x;
moverPosition.y := PositionSet.y;
moverPosition.c := PositionSet.c;

//Get Pos on track in mm
fPositionOnTrack := iTrack.PlanarTrack.GetArcLengthClosestTo(geometry:=moverPosition);

//Convert pos on track in XY
iTrack.PlanarTrack.GetPositionAt(arcLength := fPositionOnTrack, position:=trackPosition);

//Get distance to mover
DistToTrack := SQRT(EXPT((trackPosition.x - moverPosition.x),2)+EXPT((trackPosition.y - moverPosition.y),2));
END_METHOD

PROPERTY DynConstraint : REFERENCE TO DynamicConstraint_Container
GET
DynConstraint REF= THIS^.fbDynConstraintContainer;
END_GET
END_PROPERTY

METHOD Enable : HRESULT
VAR_INPUT
END_VAR
IF NOT THIS^.fbFeedback.Busy THEN
	THIS^.eActiveCommand 				:= CHALET_NC.E_NcAxisCommands.Enable;
	THIS^.fbFeedback.ActiveCommand 		:= TO_STRING(THIS^.eActiveCommand);	
	THIS^.fbFeedback.LastCommandAccepted:= TRUE;		
	THIS^.fbFeedback.Busy 				:= TRUE;

	THIS^.fbMover.Enable(fbFeedbackEnable);
	Enable := S_OK;
ELSE
	Enable := S_FALSE;
	THIS^.fbFeedback.LastCommandAccepted:= FALSE;	
END_IF
END_METHOD

{attribute 'monitoring':='call'}
//operational and position control active(hovering)
PROPERTY Enabled : BOOL
GET
(* StateDWord bit 20 - operational and position control active *)
Enabled :=  (THIS^.fbMover.MCTOPLC.STD.State = MC_PLANAR_STATE.Enabled) OR
			(THIS^.fbMover.MCTOPLC.STD.State = MC_PLANAR_STATE.Enabling) OR
			(THIS^.fbMover.MCTOPLC.STD.State = MC_PLANAR_STATE.Resetting AND PositionSet.z > 0.0) OR
			(THIS^.fbMover.MCTOPLC.STD.State = MC_PLANAR_STATE.Error AND PositionSet.z > 0.0) OR
			(THIS^.fbMover.MCTOPLC.STD.State = MC_PLANAR_STATE.ErrorPending AND PositionSet.z > 0.0) OR
			(THIS^.fbMover.MCTOPLC.STD.State = MC_PLANAR_STATE.Invalid AND PositionSet.z > 0.0);
END_GET
END_PROPERTY

METHOD FB_init : BOOL
VAR_INPUT
	bInitRetains : BOOL; // if TRUE, the retain variables are initialized (warm start / cold start)
	bInCopyCode : BOOL;  // if TRUE, the instance afterwards gets moved into the copy code (online change)
	
	
	ipSystem : I_CH_Object;
END_VAR
//Do the following code once during start up and not during onlinechange
IF NOT bInCopyCode THEN 
	
	
	(* Register to the Xplanar System
	   1. Test if the interface exists
	   2. Test if the object implements a "System for Mover" interface 
	*)
	IF ipSystem <> 0 AND_THEN __QUERYINTERFACE(ipSystem,THIS^.ipXpSystem) THEN
		THIS^.ipXpSystem.RegisterMover(THIS^);
	END_IF

	
	
	THIS^.fbFeedback.ActiveCommand 		:= TO_STRING(THIS^.eActiveCommand);	
	
	
END_IF
END_METHOD

{attribute 'monitoring':='call'}
PROPERTY Feedback : I_XP_Feedback
GET
Feedback := THIS^.fbFeedback;
END_GET
END_PROPERTY

METHOD Halt : HRESULT
VAR_INPUT
END_VAR
THIS^.eActiveCommand 				:= CHALET_NC.E_NcAxisCommands.Halt;
THIS^.fbFeedback.ActiveCommand 		:= TO_STRING(THIS^.eActiveCommand);	
THIS^.fbFeedback.LastCommandAccepted:= TRUE;		
THIS^.fbFeedback.Busy 				:= TRUE;

THIS^.fbMover.Halt(	commandFeedback := THIS^.fbFeedbackHalt, 
					constraint 		:= THIS^.fbDynConstraintContainer 
				   );

Halt := S_OK;
END_METHOD

METHOD Initialize : HRESULT
VAR
	bWaitForAxisInit : BOOL;
	hrExtAxis : HRESULT;
	stVarInfo : __SYSTEM.VAR_INFO;
	
	nIdxXpu : UDINT;
	nIdxMover : UDINT;
	ipTcIoXpu : I_TcIoXPlanarProcessingUnit;	
	//nMoverOID : OTCID;
	nOidHardwareMover : OTCID;
	hr : HRESULT;
	ipComObject : ITComObject;
	nParaSize : UDINT;
	pParaData : PVOID;
END_VAR
VAR CONSTANT
	N_IDX_HARDWARE_MOVER_OID 	: UDINT := 16#0503012D; // Parameter(online) "Hardware mover OTCID"
END_VAR

VAR_INST
	//This error cannot be reset. Requires a reset cold
	{attribute 'hide'}	
	fbInitError : FB_TcAlarm;
END_VAR
// Check if link to MC-Mover is mapped
IF NOT THIS^.Mapped THEN
	IF NOT fbInitError.bRaised THEN 
		//This error cannot be reset. Requires a reset cold
		fbInitError.CreateEx(stEventEntry:=TC_EVENTS.CHALET_Base_Events.VariableLinkMissing, ipSourceInfo := THIS^.fbSourceInfo, bWithConfirmation := FALSE);
		stVarInfo := __VARINFO(fbMover);
		fbInitError.ipArguments.AddString(stVarInfo.Symbol);
		fbInitError.Raise(0);
	END_IF
	Initialize := E_FAIL;
	RETURN;
END_IF


	
IF NOT bInitDone THEN
	//Get MC-Mover interface to utiliy lib
	FOR nIdxMover := 1 TO ipXpSystem.Enviroment.UtilityEnvirement.P_MoverCount DO
		IF ipXpSystem.Enviroment.UtilityEnvirement.P_MoverOids[nIdxMover] = THIS^.fbMover.MCTOPLC.STD.MoverOID THEN
			THIS^.ipMcMover := ipXpSystem.Enviroment.UtilityEnvirement.McMover(nIdxMover);
			EXIT;
		END_IF
	END_FOR

	
	//get OID of to MC-Mover mapped TcIoMover
	hr := FW_ObjMgr_GetObjectInstance(oid:= THIS^.fbMover.MCTOPLC.STD.MoverOID, iid:= TC_GLOBAL_IID_LIST.IID_ITComObject, pipUnk:= ADR(ipComObject));
	IF ipComObject <> 0 THEN
		//Get ADR and SIZE
		nParaSize := SIZEOF(nOidHardwareMover);	pParaData := ADR(nOidHardwareMover);
		hr := ipComObject.TcGetObjPara(pid:=N_IDX_HARDWARE_MOVER_OID , nData:= nParaSize, pData:= pParaData, pgp:=0 );
		FW_SafeRelease(ADR(ipComObject));
		
		IF nOidHardwareMover = 0 THEN
			//TODO Errormessage. MC is not mapped to TcIO
			RETURN;
		END_IF
	
		//Search interface for this OID
		FOR nIdxXpu := 1 TO ipXpSystem.Enviroment.UtilityEnvirement.P_XpuCount DO
			ipTcIoXpu := ipXpSystem.Enviroment.UtilityEnvirement.TcIoXpu(nIdxXpu);
			
			IF ipTcIoXpu <> 0 THEN
				//Get TcIo-Mover interface to utiliy lib
				FOR nIdxMover := 1 TO Param_TcIoXPlanarEnvironment.MaxXPlanarMoversPerXpu DO
					IF ipTcIoXpu.P_MoverOids[nIdxMover] = nOidHardwareMover THEN
						THIS^.ipTcIoMover := ipTcIoXpu.TcIoMover(nIdxMover);
						EXIT;
					END_IF
				END_FOR
			END_IF
		END_FOR	
	END_IF
	
	IF THIS^.ipTcIoMover = 0 OR THIS^.ipMcMover = 0 THEN
		//TODO Errormessage. Utility interface not found
		RETURN;
	END_IF
	

	//Set all move dynamic constraint to the axis default value.
	THIS^.SetDynConstraint_X(MC_DEFAULT,MC_DEFAULT,MC_DEFAULT,MC_DEFAULT);
	THIS^.SetDynConstraint_Y(MC_DEFAULT,MC_DEFAULT,MC_DEFAULT,MC_DEFAULT);	
	THIS^.SetDynConstraint_Z(MC_DEFAULT,MC_DEFAULT,MC_DEFAULT,MC_DEFAULT);	
	THIS^.SetDynConstraint_A(MC_DEFAULT,MC_DEFAULT,MC_DEFAULT,MC_DEFAULT);	
	THIS^.SetDynConstraint_B(MC_DEFAULT,MC_DEFAULT,MC_DEFAULT,MC_DEFAULT);
	THIS^.SetDynConstraint_C(MC_DEFAULT,MC_DEFAULT,MC_DEFAULT,MC_DEFAULT);
	THIS^.SetDynConstraint_Path(MC_DEFAULT,MC_DEFAULT,MC_DEFAULT,MC_DEFAULT);

	//Call Init of Setpointaxis only, if mapped
	IF AxisSetpointX.Mapped THEN hrExtAxis := GetMostSignificant(hrExtAxis, AxisSetpointX.Initialize());END_IF
	IF AxisSetpointY.Mapped THEN hrExtAxis := GetMostSignificant(hrExtAxis, AxisSetpointY.Initialize());END_IF
	IF AxisSetpointZ.Mapped THEN hrExtAxis := GetMostSignificant(hrExtAxis, AxisSetpointZ.Initialize());END_IF
	IF AxisSetpointA.Mapped THEN hrExtAxis := GetMostSignificant(hrExtAxis, AxisSetpointA.Initialize());END_IF
	IF AxisSetpointB.Mapped THEN hrExtAxis := GetMostSignificant(hrExtAxis, AxisSetpointB.Initialize());END_IF
	IF AxisSetpointC.Mapped THEN hrExtAxis := GetMostSignificant(hrExtAxis, AxisSetpointC.Initialize());END_IF	
	
	bInitDone := (hrExtAxis = S_OK);	
	
	
	//Pending
	Initialize := S_PENDING;;	
ELSE	
	//Done
	Initialize := S_OK;	
END_IF


THIS^.eActiveCommand 				:= CHALET_NC.E_NcAxisCommands.Initialize;
THIS^.fbFeedback.ActiveCommand 		:= TO_STRING(THIS^.eActiveCommand);	
THIS^.fbFeedback.LastCommandAccepted:= TRUE;	
//Set done or keep in busy state	
THIS^.fbFeedback.HR := Initialize;
END_METHOD

METHOD JoinTrack : HRESULT
VAR_INPUT
	iTrack : I_XP_Track;
END_VAR
VAR
	joinTrackOptions : ST_JoinTrackOptions;
END_VAR
IF iTrack <> 0 THEN
	THIS^.eActiveCommand 				:= CHALET_NC.E_NcAxisCommands.JoinTrack;
	THIS^.fbFeedback.ActiveCommand 		:= TO_STRING(THIS^.eActiveCommand);	
	THIS^.fbFeedback.LastCommandAccepted:= TRUE;		
	THIS^.fbFeedback.Busy 				:= TRUE;

	
	(* ADS Error 33164 or 33154: Position out of modulo range or Software position limit violation. Position must be larger or equal to zero and less or equal to the modulus when using modulo positioning. 
		When using modulo positioning, the target position is interpreted in consideration of the AdditionalTurns variable at the Options input.

		If the above error occurs, then the mover wants to rotate on the track when joining because ‘useOrientation = TRUE’ is set. 
		Better do not to set this to false, because CA then requires a much greater distance to the neighbouring mover.
		It is better to check the set C-axis modules in the MC3 PlanarMover if 90, 180 or 360°.
	*)
	joinTrackOptions.useOrientation 	:= TRUE;

	
	THIS^.fbMover.JoinTrack(commandFeedback	:= THIS^.fbFeedbackJoinTrack, 
								targetTrack	:= iTrack.PlanarTrack, 
								constraint	:= THIS^.fbDynConstraintContainer,
								options		:= joinTrackOptions);								
	JoinTrack := S_OK;
ELSE
	JoinTrack := S_FALSE;
	THIS^.fbFeedback.LastCommandAccepted:= FALSE;	
END_IF
END_METHOD

{attribute 'monitoring':='call'}
(* Retruns lentgh of hypotenuse of the x and y error. (>=0[mm]) *)
PROPERTY LagDistanceXY : LREAL
GET
VAR
	fErrorX, fErrorY : LREAL;
END_VAR
// Set - Act
fErrorX := THIS^.fbMover.MCTOPLC.SET.SetPos.X - THIS^.fbMover.MCTOPLC.ACT.ActPos.X;
fErrorY := THIS^.fbMover.MCTOPLC.SET.SetPos.Y - THIS^.fbMover.MCTOPLC.ACT.ActPos.Y;


//Dist to center. Phytagoras -> c = sqrt( A^2 + B^2)
LagDistanceXY := SQRT(EXPT(fErrorX,2) + EXPT(fErrorY,2));
END_GET
END_PROPERTY

{attribute 'monitoring':='call'}
//The last driving command given had the following value
PROPERTY LastCmdTargetGap : LREAL
GET
LastCmdTargetGap := fLastCmdTargetGap;
END_GET
END_PROPERTY

{attribute 'monitoring':='call'}
//The last driving command given had the following value
PROPERTY LastCmdTargetPosition : LREAL
GET
LastCmdTargetPosition := fLastCmdTargetPosition;
END_GET
END_PROPERTY

{attribute 'monitoring':='call'}
//The last driving command given had the following value
PROPERTY LastCmdTargetTrack: I_XP_Track
GET
LastCmdTargetTrack := ipLastCmdTrack;
END_GET
END_PROPERTY

{attribute 'monitoring':='call'}
//This was the last valid (system enabled) parent station of the mover
PROPERTY LastValidParentStation : I_XP_Station;
GET
VAR_INST

END_VAR
LastValidParentStation := THIS^.ipLastValidParentStation;
END_GET
END_PROPERTY

{attribute 'monitoring':='call'}
//This was the last valid (system enabled) actual  position of the mover
PROPERTY LastValidPositionOnTrack : LREAL
GET
VAR_INST

END_VAR
LastValidPositionOnTrack := THIS^.fLastValidPositionOnTrack;
END_GET
END_PROPERTY

{attribute 'monitoring':='call'}
//This was the last valid (system enabled) actual  position of the mover
PROPERTY LastValidPositionXYZABC : REFERENCE TO MoverVector
GET
VAR_INST

END_VAR
LastValidPositionXYZABC REF= THIS^.stLastValidPositionXYZABC;
END_GET
END_PROPERTY

{attribute 'monitoring':='call'}
//This was the last valid (system enabled) actual  position of the mover
PROPERTY LastValidTrack : I_XP_Track;
GET
VAR_INST

END_VAR
LastValidTrack := THIS^.ipLastValidTrack;
END_GET
END_PROPERTY

//The mover returns to its SetPos. The force of the Z, A and B axis is slowly increased.
METHOD LiftFromUnknownLevel : HRESULT
VAR_INPUT
END_VAR
THIS^.eActiveCommand 				:= CHALET_NC.E_NcAxisCommands.LiftFromUnknownLevel;
THIS^.fbFeedback.ActiveCommand 		:= TO_STRING(THIS^.eActiveCommand);		
THIS^.fbFeedback.Busy 				:= TRUE;


IF THIS^.fbMover.MCTOPLC.STD.State <> MC_PLANAR_STATE.Enabled THEN
	//Error wrong state
	
	;//zzz Todo Error message
	
ELSIF NOT THIS^.Standstill THEN
	//Error not allowed if mover is moving
	
	;//zzz Todo Error message
	
ELSE
	//Start of internal sequence
	THIS^.fbFeedbackLiftFromUnknown.Busy		:= TRUE;
	THIS^.nSeqLiftFromUnknown := 1;
	THIS^.nSeqLowerToUnknown := 0;
END_IF



LiftFromUnknownLevel := S_OK;
END_METHOD

(* The mover is lowered. The target height is unknown. The force from the Z, A and B axles is then reduced to a minimum. X, Y and C still remain active.
   This function can be used, for example, to place the mover in a holder.  *)
METHOD LowerToUnknownLevel : HRESULT
VAR_INPUT
END_VAR
THIS^.eActiveCommand 				:= CHALET_NC.E_NcAxisCommands.LowerToUnknownLevel;
THIS^.fbFeedback.ActiveCommand 		:= TO_STRING(THIS^.eActiveCommand);		
THIS^.fbFeedback.Busy 				:= TRUE;


IF THIS^.fbMover.MCTOPLC.STD.State <> MC_PLANAR_STATE.Enabled THEN
	//Error wrong state
	
	;//zzz Todo Error message

ELSIF NOT THIS^.Standstill THEN
	//Error not allowed if mover is moving
	
	;//zzz Todo Error message
	
	
ELSE
	//Start of internal sequence
	THIS^.fbFeedbackLowerToUnknown.Busy		:= TRUE;
	THIS^.nSeqLowerToUnknown := 1;
	THIS^.nSeqLiftFromUnknown := 0;
END_IF



LowerToUnknownLevel := S_OK;
END_METHOD

{attribute 'monitoring':='call'}
PROPERTY Mapped : BOOL //Project is mapped to MC (McToPlc and PlcToMc)
GET
VAR
	bMcToPlcNotMapped 	: BOOL;
	bPlcToMcNotMapped 	: BOOL;
END_VAR
//F_GetMappingStatus is not working on IO Data Pointer
	//bPlcToMcNotMapped := F_GetMappingStatus(ADR(THIS^.fbMover.PlcToMc), SIZEOF(THIS^.fbMover.PlcToMc)) <> EPlcMappingStatus.MS_Mapped;
	//bMcToPlcNotMapped := F_GetMappingStatus(ADR(THIS^.fbMover.McToPlc), SIZEOF(THIS^.fbMover.McToPlc)) <> EPlcMappingStatus.MS_Mapped;

	
Mapped := THIS^.fbMover.MCTOPLC.STD.MoverOID <> 0;
END_GET
END_PROPERTY

{attribute 'monitoring':='call'}
PROPERTY Mode : MC_PLANAR_MOVER_COMMAND_MODE
GET
Mode := THIS^.fbMover.MCTOPLC.STD.CommandMode;
END_GET
END_PROPERTY

METHOD MoveA : HRESULT
VAR_INPUT
	fPosition : LREAL;
END_VAR
THIS^.eActiveCommand 				:= CHALET_NC.E_NcAxisCommands.MoveA;
THIS^.fbFeedback.ActiveCommand 		:= TO_STRING(THIS^.eActiveCommand);	
THIS^.fbFeedback.LastCommandAccepted:= TRUE;		
THIS^.fbFeedback.Busy 				:= TRUE;

THIS^.fbMover.MoveA(commandFeedback	:= THIS^.fbFeedbackMoveA, 
					targetPosition	:= fPosition, 
					constraint		:= THIS^.fbDynConstraintContainer
					);

MoveA := S_OK;
END_METHOD

METHOD MoveB : HRESULT
VAR_INPUT
	fPosition : LREAL;
END_VAR
THIS^.eActiveCommand 				:= CHALET_NC.E_NcAxisCommands.MoveB;
THIS^.fbFeedback.ActiveCommand 		:= TO_STRING(THIS^.eActiveCommand);	
THIS^.fbFeedback.LastCommandAccepted:= TRUE;		
THIS^.fbFeedback.Busy 				:= TRUE;

THIS^.fbMover.MoveB(commandFeedback	:= THIS^.fbFeedbackMoveB, 
					targetPosition	:= fPosition, 
					constraint		:= THIS^.fbDynConstraintContainer
					);

MoveB := S_OK;
END_METHOD

METHOD MoveC : HRESULT
VAR_INPUT
	fPosition : LREAL;
	
	(* Addition turns to move in modulo movement (positive or negative). *)
	additionalTurns : UDINT := 0;
	
	(* Direction in which the target is approached. *)
	direction : Tc3_Mc3Definitions.MC_DIRECTION := Tc3_Mc3Definitions.MC_DIRECTION.mcDirectionNonModulo;
END_VAR
VAR
	stMoveCOptions : ST_MoveCOptions;
END_VAR
THIS^.eActiveCommand 				:= CHALET_NC.E_NcAxisCommands.MoveC;
THIS^.fbFeedback.ActiveCommand 		:= TO_STRING(THIS^.eActiveCommand);	
THIS^.fbFeedback.LastCommandAccepted:= TRUE;		
THIS^.fbFeedback.Busy 				:= TRUE;


stMoveCOptions.additionalTurns := additionalTurns;
stMoveCOptions.direction := direction;


THIS^.fbMover.MoveC(commandFeedback	:= THIS^.fbFeedbackMoveC, 
					targetPosition	:= fPosition, 
					constraint		:= THIS^.fbDynConstraintContainer, 
					options			:= stMoveCOptions
					);

MoveC := S_OK;
END_METHOD

METHOD MoveOnTrack : HRESULT
VAR_INPUT
	ipTrack : I_XP_Track;
	fPosition : LREAL;
	fGap : LREAL;
END_VAR

VAR
	moveOptions: ST_MoveOnTrackOptions;
	//fMoverDiagonal : LREAL;
END_VAR
moveOptions.direction := Tc3_Mc3Definitions.MC_DIRECTION.mcDirectionPositive;
moveOptions.additionalTurns := 0;
moveOptions.gap := XPlanarParameterlist.N_GAP_MODE_ON_TRACK; 

//Use fix gap if requested gap is to small
moveOptions.gap := MAX(fGap, XPlanarParameterlist.F_MOVER_MINIMUM_GAP_ON_TRACK);
moveOptions.dynamicMode := XPlanarParameterlist.N_SELECT_MODE_HOW_DYNAMIC_IS_PLANED_ON_TRACK;

IF ipTrack <> 0 THEN
	THIS^.eActiveCommand 				:= CHALET_NC.E_NcAxisCommands.MoveOnTrack;
	THIS^.fbFeedback.ActiveCommand 		:= TO_STRING(THIS^.eActiveCommand);	
	THIS^.fbFeedback.LastCommandAccepted:= TRUE;		
	THIS^.fbFeedback.Busy 				:= TRUE;

	THIS^.fbMover.MoveOnTrack(
		commandFeedback			:= THIS^.fbFeedbackMoveOnTrack,
		targetTrack				:= ipTrack.PlanarTrack, 
		targetPositionOnTrack	:= fPosition, 
		constraint				:= THIS^.fbDynConstraintPath, 
		options					:= moveOptions);
	
	//Store the values
	fLastCmdTargetPosition 	:= fPosition; //the last commanded target position [mm]
	fLastCmdTargetGap 		:= moveOptions.gap; //the last commanded target gap
	ipLastCmdTrack		 	:= ipTrack; //the last commanded target track	
	
	
	MoveOnTrack := S_OK;
ELSE
	MoveOnTrack := S_FALSE;
	THIS^.fbFeedback.LastCommandAccepted:= FALSE;	
END_IF
END_METHOD

METHOD MoveOnTrack_ShortestWay : HRESULT
VAR_INPUT
	ipTrack : I_XP_Track;
	fPosition : LREAL;
	fGap : LREAL;
END_VAR

VAR
	moveOptions: ST_MoveOnTrackOptions;
	//fMoverDiagonal : LREAL;
END_VAR
moveOptions.direction := Tc3_Mc3Definitions.MC_DIRECTION.mcDirectionShortestWay;
moveOptions.additionalTurns := 0;
moveOptions.gap := XPlanarParameterlist.N_GAP_MODE_ON_TRACK; 

//Use fix gap if requested gap is to small
moveOptions.gap := MAX(fGap, XPlanarParameterlist.F_MOVER_MINIMUM_GAP_ON_TRACK);
moveOptions.dynamicMode := XPlanarParameterlist.N_SELECT_MODE_HOW_DYNAMIC_IS_PLANED_ON_TRACK;

IF ipTrack <> 0 THEN
	THIS^.eActiveCommand 				:= CHALET_NC.E_NcAxisCommands.MoveOnTrack;		
	THIS^.fbFeedback.ActiveCommand 		:= TO_STRING(THIS^.eActiveCommand);	
	THIS^.fbFeedback.LastCommandAccepted:= TRUE;		
	THIS^.fbFeedback.Busy 				:= TRUE;
	
	THIS^.fbMover.MoveOnTrack(
		commandFeedback			:= THIS^.fbFeedbackMoveOnTrack,
		targetTrack				:= ipTrack.PlanarTrack, 
		targetPositionOnTrack	:= fPosition, 
		constraint				:= THIS^.fbDynConstraintPath, 
		options					:= moveOptions);
				
	fLastCmdTargetPosition 	:= fPosition; //the last commanded target position [mm]
	fLastCmdTargetGap 		:= moveOptions.gap; //the last commanded target gap
	ipLastCmdTrack		 	:= ipTrack; //the last commanded target track	
		
	MoveOnTrack_ShortestWay := S_OK;
ELSE
	MoveOnTrack_ShortestWay := S_FALSE;
	THIS^.fbFeedback.LastCommandAccepted:= FALSE;	
END_IF
END_METHOD

METHOD MoveOnTrackToStation : HRESULT
VAR_INPUT
	ipStation : I_XP_Station;
	fGap : LREAL;
END_VAR
IF ipStation <> 0 AND_THEN ipStation.AccocietedTrack <> 0 THEN

	MoveOnTrackToStation := MoveOnTrack(ipTrack:= ipStation.AccocietedTrack, 
										fPosition:= ipStation.PositionOnTrack, 
										fGap:= fGap);
ELSE
	MoveOnTrackToStation := E_FAIL;
	THIS^.fbFeedback.LastCommandAccepted:= FALSE;	
END_IF
END_METHOD

{attribute 'monitoring':='call'}
(* Height that is used for internal collision checks.[mm] *)
PROPERTY MoverHeight : LREAL
GET
VAR
	ipTrackComObject : ITComObject;
	nParaSize : UDINT;
	pParaData : PVOID;
	hr : HRESULT;
	fData : LREAL;
END_VAR
VAR CONSTANT
	N_IDX_OFFSET 	: UDINT := 16#050300B3; // Parameter(init) Mover
END_VAR
FW_ObjMgr_GetObjectInstance(oid:= THIS^.OID, iid:= TC_GLOBAL_IID_LIST.IID_ITComObject, pipUnk:= ADR(ipTrackComObject));

IF ipTrackComObject = 0 THEN
	// Error
	RETURN;
END_IF


nParaSize := SIZEOF(fData);	pParaData := ADR(fData);

hr := ipTrackComObject.TcGetObjPara(pid:=N_IDX_OFFSET , nData:= nParaSize, pData:= pParaData, pgp:=0 );
FW_SafeRelease(ADR(ipTrackComObject));


MoverHeight := fData;
END_GET
END_PROPERTY

{attribute 'monitoring':='call'}
//Mover could not be detected or was removed from the system
PROPERTY MoverIsNotPresent : BOOL
GET
VAR
	bMoverAtZeroPos, bMoverPositionInvalid, bMoverVeloInvalid : BOOL;
END_VAR
bMoverAtZeroPos		:=  PlanarMover.MCTOPLC.ACT.ActPos.x = 0 AND
						PlanarMover.MCTOPLC.ACT.ActPos.y = 0 AND 
						PlanarMover.MCTOPLC.ACT.ActPos.z = 0 AND 
						PlanarMover.MCTOPLC.ACT.ActPos.a = 0 AND
						PlanarMover.MCTOPLC.ACT.ActPos.b = 0 AND 
						PlanarMover.MCTOPLC.ACT.ActPos.c = 0 AND 
						PlanarMover.MCTOPLC.ACT.PhysicalAreaID = 0;
						
						
bMoverPositionInvalid:=  PlanarMover.MCTOPLC.ACT.ActPos.x >= 1E+302 AND
						PlanarMover.MCTOPLC.ACT.ActPos.y >= 1E+302 AND 
						PlanarMover.MCTOPLC.ACT.ActPos.z >= 1E+302 AND 
						PlanarMover.MCTOPLC.ACT.ActPos.a >= 1E+302 AND
						PlanarMover.MCTOPLC.ACT.ActPos.b >= 1E+302 AND 
						PlanarMover.MCTOPLC.ACT.ActPos.c >= 1E+302;
						
						
bMoverVeloInvalid	:=  PlanarMover.MCTOPLC.ACT.ActVelo.x >= 1E+302 AND
						PlanarMover.MCTOPLC.ACT.ActVelo.y >= 1E+302 AND 
						PlanarMover.MCTOPLC.ACT.ActVelo.z >= 1E+302 AND 
						PlanarMover.MCTOPLC.ACT.ActVelo.a >= 1E+302 AND
						PlanarMover.MCTOPLC.ACT.ActVelo.b >= 1E+302 AND 
						PlanarMover.MCTOPLC.ACT.ActVelo.c >= 1E+302;
						
MoverIsNotPresent := bMoverAtZeroPos OR bMoverPositionInvalid OR bMoverVeloInvalid;
END_GET
END_PROPERTY

{attribute 'monitoring':='call'}
(* Width that is used for internal collision checks.[mm] *)
PROPERTY MoverWidth : LREAL
GET
VAR
	ipTrackComObject : ITComObject;
	nParaSize : UDINT;
	pParaData : PVOID;
	hr : HRESULT;
	fData : LREAL;
END_VAR
VAR CONSTANT
	N_IDX_OFFSET 	: UDINT := 16#050300B2; // Parameter(init) Mover
END_VAR
FW_ObjMgr_GetObjectInstance(oid:= THIS^.OID, iid:= TC_GLOBAL_IID_LIST.IID_ITComObject, pipUnk:= ADR(ipTrackComObject));

IF ipTrackComObject = 0 THEN
	// Error
	RETURN;
END_IF


nParaSize := SIZEOF(fData);	pParaData := ADR(fData);
hr := ipTrackComObject.TcGetObjPara(pid:=N_IDX_OFFSET , nData:= nParaSize, pData:= pParaData, pgp:=0 );
FW_SafeRelease(ADR(ipTrackComObject));

MoverWidth := fData;
END_GET
END_PROPERTY

METHOD MoveXY : HRESULT
VAR_INPUT
	fPosition_X : LREAL;
	fPosition_Y : LREAL;
END_VAR
VAR
	fbTargetPosition 	: PositionXYC;
	stMoveOptions 		: ST_MoveToPositionOptions;
END_VAR
THIS^.eActiveCommand 				:= CHALET_NC.E_NcAxisCommands.MoveXY;
THIS^.fbFeedback.ActiveCommand 		:= TO_STRING(THIS^.eActiveCommand);	
THIS^.fbFeedback.LastCommandAccepted:= TRUE;		
THIS^.fbFeedback.Busy 				:= TRUE;



fbTargetPosition.SetValuesXY(x := fPosition_X, y := fPosition_Y);

stMoveOptions.useOrientation := TRUE;

THIS^.fbMover.MoveToPosition(	commandFeedback	:= THIS^.fbFeedbackMoveXY, 
								targetPosition	:= fbTargetPosition,
								constraint		:= THIS^.fbDynConstraintContainer, 
								options			:= stMoveOptions);

MoveXY := S_OK;
END_METHOD

METHOD MoveZ : HRESULT
VAR_INPUT
	fPosition : LREAL;
END_VAR
THIS^.eActiveCommand 				:= CHALET_NC.E_NcAxisCommands.MoveZ;
THIS^.fbFeedback.ActiveCommand 		:= TO_STRING(THIS^.eActiveCommand);	
THIS^.fbFeedback.LastCommandAccepted:= TRUE;		
THIS^.fbFeedback.Busy 				:= TRUE;


THIS^.fbMover.MoveZ(commandFeedback	:= THIS^.fbFeedbackMoveZ, 
					targetPosition	:= fPosition, 
					constraint		:= THIS^.fbDynConstraintContainer
					);

MoveZ := S_OK;
END_METHOD

{attribute 'monitoring':='call'}
//Unique object ID
PROPERTY OID : OTCID
GET
OID := THIS^.fbMover.MCTOPLC.STD.MoverOID;
END_GET
END_PROPERTY

{attribute 'monitoring':='call'}
PROPERTY ParentStation : I_XP_Station
GET
ParentStation := ipParentStation;
END_GET
SET
THIS^.ipParentStation := ParentStation;

IF ParentStation <> 0 THEN
	THIS^.ipLastValidParentStation := ParentStation;
END_IF
END_SET
END_PROPERTY

{attribute 'monitoring':='call'}
PROPERTY PlanarMover : REFERENCE TO MC_PlanarMover
GET
PlanarMover ref= THIS^.fbMover;
END_GET
END_PROPERTY

{attribute 'monitoring':='call'}
(* Contains the information of the Planar Mover passed from MC to PLC. XYZABC [mm] *)
PROPERTY PositionAct : REFERENCE TO MoverVector
GET
VAR_INST
	{attribute 'hide'}
	copyOfActPosition :  MoverVector;
END_VAR
//Creat an copy of the struct to view value in targetdbrowser and plc online view
copyOfActPosition := THIS^.fbMover.MCTOPLC.ACT.ActPos;
PositionAct REF= copyOfActPosition;
END_GET
END_PROPERTY

{attribute 'monitoring':='call'}
PROPERTY PositionOnTrack : LREAL
GET
VAR_INST
	{attribute 'hide'}	
	fPosOnTrack : LREAL;
END_VAR
fPosOnTrack := THIS^.fbMover.MCTOPLC.SETONTRACK.SetPos;
PositionOnTrack := fPosOnTrack;
END_GET
END_PROPERTY

{attribute 'monitoring':='call'}
(* Provides the current planar mover setpoint XYZABC [mm] *)
PROPERTY PositionSet : REFERENCE TO MoverVector
GET
VAR_INST
	{attribute 'hide'}
	copyOfSetPosition :  MoverVector;
END_VAR
//Creat an copy of the struct to view value in targetdbrowser and plc online view
copyOfSetPosition := THIS^.fbMover.MCTOPLC.SET.SetPos;
PositionSet REF= copyOfSetPosition;
END_GET
END_PROPERTY

(* Time-critical information is processed here, which can then be polled via the property every cycle. 
The update method is usually at the end of the program and then it is already 'outdated'. *)
METHOD PRIVATE Prepare : HRESULT
VAR

END_VAR
VAR_INST
	{attribute 'hide'}
	nLastUpdatedCycleCount : UDINT;
END_VAR
//Check if this Cycle the dates are allready prepared
IF nLastUpdatedCycleCount <> TwinCAT_SystemInfoVarList._TaskInfo[THIS^.nTaskIndex].CycleCount THEN
	nLastUpdatedCycleCount := TwinCAT_SystemInfoVarList._TaskInfo[THIS^.nTaskIndex].CycleCount;

	//Stor last valide position im system is enabled
	IF ipXpSystem.Enabled THEN
		THIS^.stLastValidPositionXYZABC := THIS^.PositionSet;
		THIS^.fLastValidPositionOnTrack := THIS^.PositionOnTrack;
		THIS^.ipLastValidTrack := THIS^.CurrentTrack;
	END_IF

END_IF
END_METHOD

{attribute 'monitoring':='call'}
PROPERTY PUBLIC ProductData : I_XP_ProductData
GET
ProductData := ipProductData;
END_GET
SET
// No change. Same interface is set again
IF ipProductData = ProductData THEN
	;//Noting
	
ELSE

	// If allready an interface is linked. Unlink
	IF ipProductData <> 0 THEN
		ipProductData.LinkToMover(0);
		ipProductData := 0;
	END_IF
	
	// Link and store new interface
	IF ProductData <> 0 THEN
		ProductData.LinkToMover(THIS^);
		ipProductData := ProductData;
	END_IF
END_IF
END_SET
END_PROPERTY

METHOD RemoveFromGroup : HRESULT

VAR
	iGroup: INT;
END_VAR
IF NOT THIS^.fbFeedback.Busy THEN
	THIS^.eActiveCommand 				:= CHALET_NC.E_NcAxisCommands.RemoveFromGroupe;
	THIS^.fbFeedback.ActiveCommand 	:= TO_STRING(THIS^.eActiveCommand);	
	THIS^.fbFeedback.LastCommandAccepted:= TRUE;		
	THIS^.fbFeedback.Busy 				:= TRUE;
	
	THIS^.fbMover.RemoveFromGroup(THIS^.fbFeedbackRmvFromGrp);
	
	RemoveFromGroup := S_OK;
ELSE
	RemoveFromGroup := S_FALSE;
	THIS^.fbFeedback.LastCommandAccepted:= FALSE;	
END_IF
END_METHOD

METHOD Reset : HRESULT
VAR_INPUT
END_VAR
THIS^.eActiveCommand 				:= CHALET_NC.E_NcAxisCommands.Reset;
THIS^.fbFeedback.ActiveCommand 		:= TO_STRING(THIS^.eActiveCommand);	
THIS^.fbFeedback.LastCommandAccepted:= TRUE;		
THIS^.fbFeedback.Busy 				:= TRUE;

THIS^.fbMover.Reset(THIS^.fbFeedbackReset);
Reset := S_OK;
END_METHOD

{attribute 'monitoring':='call'}
//Complete route from last parent to active parent station
PROPERTY RouteComplete : I_CH_List
GET
RouteComplete := THIS^.fbRouteComplete;
END_GET
END_PROPERTY

{attribute 'monitoring':='call'}
//Remaining route to the parent
PROPERTY RouteRemaining: I_CH_List
GET
RouteRemaining := THIS^.fbRouteRemaining;
END_GET
END_PROPERTY

//done segments can be transferred here. these are removed from the remaining route
METHOD RouteSegmentDone : BOOL
VAR_INPUT
	ipPathDone : I_XP_Path;
END_VAR
RouteSegmentDone := THIS^.fbRouteRemaining.RemoveObject(ipPathDone);
END_METHOD

METHOD SetDynConstraint_A : BOOL //Dynamic constraints for individual coordinates.
VAR_INPUT
    V : MC_LREAL; //equivalent to data type LREAL + MC_DEFAULT, MC_MAXIMUM
    A : MC_LREAL; //equivalent to data type LREAL + MC_DEFAULT, MC_MAXIMUM
    D : MC_LREAL; //equivalent to data type LREAL + MC_DEFAULT, MC_MAXIMUM
    J : MC_LREAL; //equivalent to data type LREAL + MC_DEFAULT, MC_MAXIMUM
END_VAR
THIS^.fbDynConstraintCoordinates.SetLimit(	Coordinate := Coord_Mcs_A1, 
											V := V, 
											A := A, 
											D := D, 
											J := J);
											
//Changes to the origin constraint do not affect the copy of the constraint in the instance of the DynamicConstraint_Container.
//For this reason, the container is being refreshed here							
fbDynConstraintContainer.Clear();
fbDynConstraintContainer.AddConstraint(fbDynConstraintPath);
fbDynConstraintContainer.AddConstraint(fbDynConstraintCoordinates);
END_METHOD

METHOD SetDynConstraint_B : BOOL //Dynamic constraints for individual coordinates.
VAR_INPUT
    V : MC_LREAL; //equivalent to data type LREAL + MC_DEFAULT, MC_MAXIMUM
    A : MC_LREAL; //equivalent to data type LREAL + MC_DEFAULT, MC_MAXIMUM
    D : MC_LREAL; //equivalent to data type LREAL + MC_DEFAULT, MC_MAXIMUM
    J : MC_LREAL; //equivalent to data type LREAL + MC_DEFAULT, MC_MAXIMUM
END_VAR
THIS^.fbDynConstraintCoordinates.SetLimit(	Coordinate := Coord_Mcs_B1, 
											V := V, 
											A := A, 
											D := D, 
											J := J);											

